KUKA KRL program: MyProgram_311().src

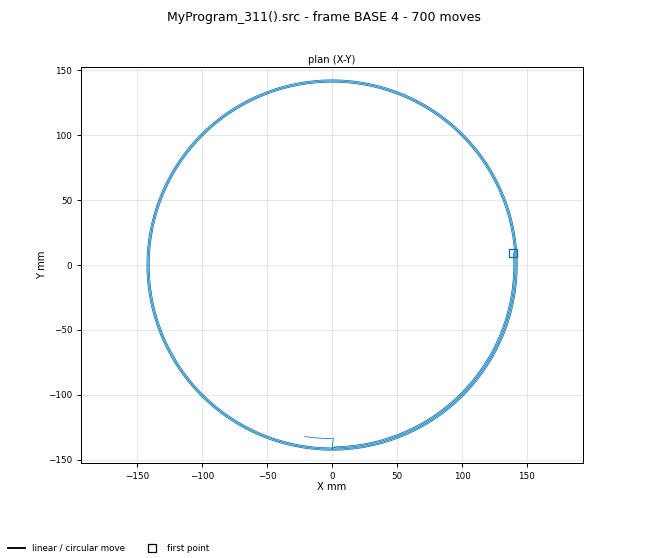
[picture p0: tool path of MyProgram_311().src in frame BASE 4, 700 of 700 moves have a stored position in this frame; points joined in program order, loops and branches not executed]
&ACCESS RVP
&REL 1
&PARAM TEMPLATE = C:\KRC\Roboter\Template\vorgabe
&PARAM EDITMASK = *
DEF MyProgram_311()
; ---- Setting reference (Base) ----
$BASE = BASE_DATA[4]

; --------------------------
; ---- Setting tool (TCP) ----
$TOOL = TOOL_DATA[3]
; --------------------------

$VEL.CP = VEL_APROX_PRINT
Startdeposition()
$VEL.CP = VEL_PRINT
LIN {X 139.5556,Y 9.3465,Z 182,A 6.1945,B 4.3682,C 0.2186,E1 4.5332,E2 446.7738} C_DIS
LIN {X 139.7636,Y 5.3586,Z 182,A 4.7306,B 4.3681,C 0.221,E1 4.5334,E2 448.2166} C_DIS
LIN {X 139.863,Y 1.0803,Z 182,A 3.0816,B 4.3679,C 0.2246,E1 4.5334,E2 449.8533} C_DIS
LIN {X 139.8455,Y -2.4148,Z 182,A 1.6288,B 4.3677,C 0.229,E1 4.5334,E2 451.3099} C_DIS
LIN {X 139.7039,Y -6.743,Z 182,A -0.0934,B 4.3674,C 0.2333,E1 4.5332,E2 453.0267} C_DIS
LIN {X 139.4575,Y -10.6969,Z 182,A -1.7087,B 4.3672,C 0.2378,E1 4.5329,E2 454.6422} C_DIS
LIN {X 139.0946,Y -14.6738,Z 182,A -3.2274,B 4.367,C 0.2409,E1 4.5325,E2 456.1468} C_DIS
LIN {X 138.7184,Y -17.8838,Z 182,A -4.5556,B 4.3668,C 0.2447,E1 4.5321,E2 457.4766} C_DIS
LIN {X 138.1883,Y -21.5997,Z 182,A -5.9216,B 4.3667,C 0.2468,E1 4.5315,E2 458.8215} C_DIS
LIN {X 137.1011,Y -27.6739,Z 182,A -8.4598,B 4.3663,C 0.254,E1 4.5302,E2 461.363} C_DIS
LIN {X 136.3972,Y -30.9569,Z 182,A -9.732,B 4.3661,C 0.2565,E1 4.5295,E2 462.6228} C_DIS
LIN {X 135.1669,Y -35.95,Z 182,A -11.6103,B 4.366,C 0.2593,E1 4.5282,E2 464.4729} C_DIS
LIN {X 133.3888,Y -42.0731,Z 182,A -14.3818,B 4.3654,C 0.2686,E1 4.526,E2 467.2676} C_DIS
LIN {X 132.1888,Y -45.7009,Z 182,A -15.8575,B 4.3652,C 0.2716,E1 4.5247,E2 468.7328} C_DIS
LIN {X 131.0744,Y -48.8061,Z 182,A -17.1041,B 4.3651,C 0.2739,E1 4.5235,E2 469.9668} C_DIS
LIN {X 129.9588,Y -51.7063,Z 182,A -18.4546,B 4.3648,C 0.2783,E1 4.5221,E2 471.3286} C_DIS
LIN {X 128.6386,Y -54.9087,Z 182,A -19.8601,B 4.3646,C 0.2819,E1 4.5206,E2 472.7336} C_DIS
LIN {X 127.1217,Y -58.3322,Z 182,A -21.2882,B 4.3644,C 0.2845,E1 4.519,E2 474.1489} C_DIS
LIN {X 125.7052,Y -61.327,Z 182,A -22.6522,B 4.3642,C 0.2881,E1 4.5173,E2 475.515} C_DIS
LIN {X 123.9954,Y -64.7123,Z 182,A -24.1146,B 4.364,C 0.2909,E1 4.5155,E2 476.9667} C_DIS
LIN {X 121.8931,Y -68.5935,Z 182,A -25.947,B 4.3637,C 0.2958,E1 4.513,E2 478.804} C_DIS
LIN {X 119.5124,Y -72.6628,Z 182,A -28.2329,B 4.363,C 0.3051,E1 4.5096,E2 481.138} C_DIS
LIN {X 117.0621,Y -76.5483,Z 182,A -29.6908,B 4.363,C 0.3043,E1 4.5075,E2 482.5419} C_DIS
LIN {X 114.3471,Y -80.5465,Z 182,A -31.6337,B 4.3628,C 0.3086,E1 4.5044,E2 484.4817} C_DIS
LIN {X 112.2761,Y -83.4091,Z 182,A -33.5934,B 4.3621,C 0.3184,E1 4.5011,E2 486.5099} C_DIS
LIN {X 108.7982,Y -87.8973,Z 182,A -35.2386,B 4.3623,C 0.3151,E1 4.4983,E2 488.0676} C_DIS
LIN {X 105.9724,Y -91.2843,Z 182,A -37.4172,B 4.3617,C 0.3238,E1 4.4943,E2 490.2968} C_DIS
LIN {X 102.9688,Y -94.6595,Z 182,A -38.9115,B 4.3617,C 0.3234,E1 4.4916,E2 491.7457} C_DIS
LIN {X 99.538,Y -98.2618,Z 182,A -40.8482,B 4.3615,C 0.3264,E1 4.4878,E2 493.6707} C_DIS
LIN {X 96.3702,Y -101.3701,Z 182,A -42.5691,B 4.3613,C 0.3289,E1 4.4844,E2 495.3802} C_DIS
LIN {X 93.176,Y -104.3133,Z 182,A -44.299,B 4.3611,C 0.3319,E1 4.4808,E2 497.105} C_DIS
LIN {X 89.7656,Y -107.262,Z 182,A -46.1268,B 4.3608,C 0.3352,E1 4.4769,E2 498.9318} C_DIS
LIN {X 86.198,Y -110.1496,Z 182,A -47.8249,B 4.3608,C 0.3365,E1 4.4733,E2 500.6072} C_DIS
LIN {X 83.8613,Y -111.9394,Z 182,A -49.0987,B 4.3605,C 0.3394,E1 4.4704,E2 501.8911} C_DIS
LIN {X 78.9883,Y -115.4291,Z 182,A -51.5583,B 4.3601,C 0.3437,E1 4.4648,E2 504.3532} C_DIS
LIN {X 76.295,Y -117.2266,Z 182,A -53.2496,B 4.3596,C 0.3503,E1 4.4607,E2 506.094} C_DIS
LIN {X 72.5505,Y -119.5803,Z 182,A -54.3551,B 4.3601,C 0.3448,E1 4.4583,E2 507.1069} C_DIS
LIN {X 67.227,Y -122.6523,Z 182,A -57.1169,B 4.3595,C 0.3515,E1 4.4515,E2 509.9034} C_DIS
LIN {X 63.5857,Y -124.5765,Z 182,A -58.5717,B 4.3595,C 0.3511,E1 4.448,E2 511.3284} C_DIS
LIN {X 60.5652,Y -126.0729,Z 182,A -60.0389,B 4.3593,C 0.354,E1 4.4443,E2 512.8082} C_DIS
LIN {X 57.3664,Y -127.5602,Z 182,A -61.391,B 4.3593,C 0.3548,E1 4.4409,E2 514.1489} C_DIS
LIN {X 54.213,Y -128.9321,Z 182,A -62.8205,B 4.3591,C 0.3568,E1 4.4372,E2 515.5822} C_DIS
LIN {X 50.9804,Y -130.2442,Z 182,A -64.1651,B 4.3591,C 0.3575,E1 4.4337,E2 516.9165} C_DIS
LIN {X 47.7376,Y -131.4674,Z 182,A -65.6245,B 4.3589,C 0.3595,E1 4.4299,E2 518.3822} C_DIS
LIN {X 44.4095,Y -132.6285,Z 182,A -67.1062,B 4.3587,C 0.3615,E1 4.426,E2 519.8699} C_DIS
LIN {X 41.0102,Y -133.7185,Z 182,A -68.4928,B 4.3587,C 0.362,E1 4.4223,E2 521.2473} C_DIS
LIN {X 37.9473,Y -134.6201,Z 182,A -69.7052,B 4.3587,C 0.3622,E1 4.4191,E2 522.4478} C_DIS
LIN {X 34.2391,Y -135.6104,Z 182,A -71.6562,B 4.3582,C 0.3677,E1 4.4136,E2 524.4505} C_DIS
LIN {X 29.2302,Y -136.7778,Z 182,A -73.4098,B 4.3584,C 0.3654,E1 4.409,E2 526.1581} C_DIS
LIN {X 23.4061,Y -137.8942,Z 182,A -75.738,B 4.3584,C 0.3659,E1 4.4027,E2 528.4743} C_DIS
LIN {X 19.0292,Y -138.5677,Z 182,A -77.8353,B 4.358,C 0.3699,E1 4.3967,E2 530.6106} C_DIS
LIN {X 15.027,Y -139.0566,Z 182,A -79.3975,B 4.358,C 0.3697,E1 4.3924,E2 532.1618} C_DIS
LIN {X 10.8973,Y -139.4429,Z 182,A -81.106,B 4.358,C 0.3705,E1 4.3877,E2 533.8725} C_DIS
LIN {X 6.9643,Y -139.6928,Z 182,A -82.6912,B 4.358,C 0.3707,E1 4.3832,E2 535.4545} C_DIS
LIN {X 2.5889,Y -139.8426,Z 182,A -84.4714,B 4.358,C 0.3709,E1 4.3783,E2 537.2339} C_DIS
LIN {X 2.5889,Y -139.8426,Z 182,A -84.4714,B 4.358,C 0.3709,E1 4.3783,E2 537.2339} C_DIS
Enddeposition()
LIN {X 1.0035,Y -140.7616,Z 182,A -84.5459,B 4.3128,C 0.3663,E1 4.3327,E2 537.2758} C_DIS
Startdeposition()
$VEL.CP = VEL_PRINT
LIN {X 4.1947,Y -140.7055,Z 182,A -83.0241,B 4.313,C 0.3637,E1 4.3371,E2 535.7232} C_DIS
LIN {X 8.4297,Y -140.5153,Z 182,A -81.3313,B 4.313,C 0.3635,E1 4.3418,E2 534.0339} C_DIS
LIN {X 12.0807,Y -140.2485,Z 182,A -79.8862,B 4.313,C 0.3635,E1 4.3458,E2 532.5942} C_DIS
LIN {X 15.6538,Y -139.8958,Z 182,A -78.4155,B 4.313,C 0.3627,E1 4.3499,E2 531.1214} C_DIS
LIN {X 21.7686,Y -139.0744,Z 182,A -75.9054,B 4.3132,C 0.3614,E1 4.3569,E2 528.6101} C_DIS
LIN {X 25.7531,Y -138.3934,Z 182,A -74.2127,B 4.3133,C 0.3599,E1 4.3615,E2 526.91} C_DIS
LIN {X 29.5156,Y -137.6385,Z 182,A -72.6715,B 4.3133,C 0.359,E1 4.3657,E2 525.3706} C_DIS
LIN {X 33.4498,Y -136.7363,Z 182,A -71.1692,B 4.3133,C 0.3593,E1 4.3698,E2 523.8865} C_DIS
LIN {X 36.5552,Y -135.9385,Z 182,A -69.7439,B 4.3136,C 0.3568,E1 4.3737,E2 522.4439} C_DIS
LIN {X 41.4818,Y -134.5169,Z 182,A -67.7824,B 4.3136,C 0.3563,E1 4.3789,E2 520.4982} C_DIS
LIN {X 44.766,Y -133.4599,Z 182,A -66.3864,B 4.3137,C 0.3549,E1 4.3826,E2 519.1023} C_DIS
LIN {X 48.3681,Y -132.1983,Z 182,A -64.8799,B 4.3138,C 0.3538,E1 4.3865,E2 517.6013} C_DIS
LIN {X 51.4087,Y -131.0449,Z 182,A -63.5613,B 4.3139,C 0.3524,E1 4.39,E2 516.2824} C_DIS
LIN {X 54.4767,Y -129.7989,Z 182,A -62.2082,B 4.3141,C 0.3507,E1 4.3935,E2 514.9276} C_DIS
LIN {X 57.7378,Y -128.3816,Z 182,A -60.7873,B 4.3141,C 0.3491,E1 4.3971,E2 513.5092} C_DIS
LIN {X 61.0166,Y -126.8563,Z 182,A -59.3503,B 4.3143,C 0.3476,E1 4.4007,E2 512.0759} C_DIS
LIN {X 64.2712,Y -125.239,Z 182,A -57.9029,B 4.3144,C 0.3459,E1 4.4043,E2 510.6317} C_DIS
LIN {X 67.2412,Y -123.6715,Z 182,A -56.2495,B 4.3149,C 0.3405,E1 4.4085,E2 508.9383} C_DIS
LIN {X 70.2583,Y -121.9829,Z 182,A -54.9598,B 4.3149,C 0.3398,E1 4.4116,E2 507.6636} C_DIS
LIN {X 74.8899,Y -119.1955,Z 182,A -53.001,B 4.3149,C 0.3392,E1 4.4161,E2 505.736} C_DIS
LIN {X 78.4114,Y -116.909,Z 182,A -50.8592,B 4.3156,C 0.3311,E1 4.4213,E2 503.5337} C_DIS
LIN {X 82.0265,Y -114.4012,Z 182,A -49.4942,B 4.3154,C 0.3332,E1 4.4243,E2 502.2254} C_DIS
LIN {X 85.449,Y -111.8679,Z 182,A -47.8119,B 4.3156,C 0.3307,E1 4.428,E2 500.5486} C_DIS
LIN {X 88.8686,Y -109.1715,Z 182,A -46.0808,B 4.3159,C 0.3279,E1 4.4318,E2 498.8218} C_DIS
LIN {X 92.2336,Y -106.3443,Z 182,A -44.3097,B 4.3161,C 0.3247,E1 4.4355,E2 497.0515} C_DIS
LIN {X 95.5139,Y -103.4078,Z 182,A -42.5311,B 4.3163,C 0.3213,E1 4.4392,E2 495.2734} C_DIS
LIN {X 98.8564,Y -100.2175,Z 182,A -40.6973,B 4.3166,C 0.318,E1 4.4429,E2 493.4443} C_DIS
LIN {X 102.055,Y -96.9583,Z 182,A -38.5045,B 4.3172,C 0.3099,E1 4.4472,E2 491.2045} C_DIS
LIN {X 105.1058,Y -93.6422,Z 182,A -37.3641,B 4.3168,C 0.3147,E1 4.4492,E2 490.1566} C_DIS
LIN {X 108.3519,Y -89.8657,Z 182,A -35.1583,B 4.3173,C 0.3079,E1 4.4532,E2 487.925} C_DIS
LIN {X 112.1364,Y -85.0962,Z 182,A -32.6312,B 4.3178,C 0.3016,E1 4.4575,E2 485.3891} C_DIS
LIN {X 116.9021,Y -78.4217,Z 182,A -29.6507,B 4.318,C 0.2983,E1 4.4623,E2 482.4542} C_DIS
LIN {X 120.7242,Y -72.4002,Z 182,A -26.7535,B 4.3185,C 0.2912,E1 4.4666,E2 479.5555} C_DIS
LIN {X 122.5931,Y -69.1878,Z 182,A -25.1638,B 4.3188,C 0.2865,E1 4.4688,E2 477.9542} C_DIS
LIN {X 124.7296,Y -65.2531,Z 182,A -23.5005,B 4.319,C 0.2839,E1 4.4709,E2 476.3106} C_DIS
LIN {X 126.4028,Y -61.9505,Z 182,A -22.0299,B 4.3192,C 0.2805,E1 4.4728,E2 474.8437} C_DIS
LIN {X 127.8752,Y -58.8507,Z 182,A -20.675,B 4.3194,C 0.2774,E1 4.4743,E2 473.4931} C_DIS
LIN {X 129.3099,Y -55.6276,Z 182,A -19.2888,B 4.3196,C 0.2743,E1 4.4759,E2 472.1125} C_DIS
LIN {X 130.5822,Y -52.5709,Z 182,A -17.97,B 4.3198,C 0.2711,E1 4.4773,E2 470.7963} C_DIS
LIN {X 131.8258,Y -49.3698,Z 182,A -16.5883,B 4.32,C 0.2675,E1 4.4787,E2 469.4156} C_DIS
LIN {X 133.0706,Y -45.9097,Z 182,A -15.1591,B 4.3202,C 0.2644,E1 4.48,E2 467.9943} C_DIS
LIN {X 134.1721,Y -42.5836,Z 182,A -13.5517,B 4.3206,C 0.2581,E1 4.4814,E2 466.3614} C_DIS
LIN {X 136.0007,Y -36.322,Z 182,A -10.8431,B 4.321,C 0.2501,E1 4.4834,E2 463.6435} C_DIS
LIN {X 136.9727,Y -32.4689,Z 182,A -9.7672,B 4.3209,C 0.2528,E1 4.4841,E2 462.6387} C_DIS
LIN {X 137.5669,Y -29.8472,Z 182,A -7.7789,B 4.3217,C 0.2379,E1 4.4853,E2 460.5298} C_DIS
LIN {X 138.7895,Y -23.5179,Z 182,A -6.228,B 4.3214,C 0.2448,E1 4.486,E2 459.1204} C_DIS
LIN {X 139.3977,Y -19.5929,Z 182,A -4.467,B 4.3217,C 0.2383,E1 4.4867,E2 457.3391} C_DIS
LIN {X 139.9332,Y -15.3061,Z 182,A -2.7578,B 4.322,C 0.234,E1 4.4873,E2 455.6351} C_DIS
LIN {X 140.3029,Y -11.4371,Z 182,A -1.2902,B 4.3221,C 0.231,E1 4.4876,E2 454.1814} C_DIS
LIN {X 140.521,Y -8.3358,Z 182,A -0.0362,B 4.3223,C 0.2276,E1 4.4879,E2 452.9281} C_DIS
LIN {X 140.7039,Y -4.2549,Z 182,A 1.6616,B 4.3226,C 0.2224,E1 4.488,E2 451.2244} C_DIS
LIN {X 140.7701,Y -0.1592,Z 182,A 3.1572,B 4.3226,C 0.2199,E1 4.488,E2 449.7503} C_DIS
LIN {X 140.7346,Y 3.1471,Z 182,A 4.6254,B 4.323,C 0.2145,E1 4.488,E2 448.2651} C_DIS
LIN {X 140.5902,Y 7.0668,Z 182,A 6.0508,B 4.323,C 0.2122,E1 4.4878,E2 446.861} C_DIS
LIN {X 140.3777,Y 10.4737,Z 182,A 7.3856,B 4.3232,C 0.209,E1 4.4876,E2 445.5325} C_DIS
LIN {X 140.018,Y 14.5186,Z 182,A 9.7771,B 4.3239,C 0.1947,E1 4.4869,E2 443.042} C_DIS
LIN {X 139.2272,Y 20.7812,Z 182,A 11.4394,B 4.3237,C 0.1994,E1 4.4863,E2 441.4984} C_DIS
LIN {X 138.7977,Y 23.4691,Z 182,A 12.566,B 4.3238,C 0.196,E1 4.4857,E2 440.3685} C_DIS
LIN {X 138.2105,Y 26.7099,Z 182,A 14.4089,B 4.3243,C 0.1857,E1 4.4847,E2 438.4585} C_DIS
LIN {X 137.1859,Y 31.5521,Z 182,A 15.8637,B 4.3243,C 0.1874,E1 4.4839,E2 437.0765} C_DIS
LIN {X 136.2457,Y 35.4009,Z 182,A 17.3501,B 4.3243,C 0.1847,E1 4.4829,E2 435.6057} C_DIS
LIN {X 135.3426,Y 38.7107,Z 182,A 18.931,B 4.3246,C 0.1785,E1 4.4817,E2 433.9998} C_DIS
LIN {X 134.0511,Y 42.9623,Z 182,A 20.4982,B 4.3246,C 0.1767,E1 4.4804,E2 432.4633} C_DIS
LIN {X 132.8883,Y 46.4356,Z 182,A 21.8914,B 4.3248,C 0.1739,E1 4.4791,E2 431.082} C_DIS
LIN {X 131.8874,Y 49.2054,Z 182,A 23.5596,B 4.3251,C 0.1647,E1 4.4774,E2 429.3517} C_DIS
LIN {X 130.1998,Y 53.5169,Z 182,A 24.8803,B 4.3251,C 0.167,E1 4.4761,E2 428.104} C_DIS
LIN {X 128.92,Y 56.5293,Z 182,A 26.1907,B 4.3251,C 0.1638,E1 4.4747,E2 426.7958} C_DIS
LIN {X 127.624,Y 59.3939,Z 182,A 27.464,B 4.3253,C 0.1606,E1 4.4732,E2 425.5227} C_DIS
LIN {X 126.0079,Y 62.7509,Z 182,A 28.92,B 4.3254,C 0.1575,E1 4.4714,E2 424.0739} C_DIS
LIN {X 124.1359,Y 66.3803,Z 182,A 30.6357,B 4.3256,C 0.1526,E1 4.4692,E2 422.3506} C_DIS
LIN {X 120.9487,Y 72.0235,Z 182,A 32.8923,B 4.3256,C 0.1509,E1 4.4661,E2 420.1425} C_DIS
LIN {X 119.5449,Y 74.3303,Z 182,A 34.2434,B 4.3258,C 0.1451,E1 4.4641,E2 418.7584} C_DIS
LIN {X 117.0756,Y 78.1618,Z 182,A 36.0299,B 4.326,C 0.1415,E1 4.4614,E2 416.9802} C_DIS
LIN {X 114.7222,Y 81.5777,Z 182,A 37.6874,B 4.326,C 0.1379,E1 4.4587,E2 415.3261} C_DIS
LIN {X 112.1161,Y 85.1241,Z 182,A 39.4657,B 4.3262,C 0.134,E1 4.4557,E2 413.549} C_DIS
LIN {X 108.7195,Y 89.4211,Z 182,A 41.7328,B 4.3264,C 0.1286,E1 4.4517,E2 411.2764} C_DIS
LIN {X 105.3023,Y 93.4208,Z 182,A 43.7256,B 4.3264,C 0.1258,E1 4.4481,E2 409.3023} C_DIS
LIN {X 102.4492,Y 96.5408,Z 182,A 45.391,B 4.3265,C 0.1228,E1 4.445,E2 407.6436} C_DIS
LIN {X 99.1559,Y 99.9204,Z 182,A 47.6585,B 4.3268,C 0.1147,E1 4.4404,E2 405.331} C_DIS
LIN {X 95.9178,Y 103.0324,Z 182,A 49.2458,B 4.3268,C 0.114,E1 4.4372,E2 403.7745} C_DIS
LIN {X 93.3927,Y 105.3272,Z 182,A 50.098,B 4.3267,C 0.1177,E1 4.4356,E2 402.9911} C_DIS
LIN {X 91.4403,Y 107.0269,Z 182,A 51.4759,B 4.3268,C 0.1119,E1 4.4326,E2 401.5716} C_DIS
LIN {X 88.5315,Y 109.4449,Z 182,A 52.9487,B 4.3268,C 0.1099,E1 4.4294,E2 400.1071} C_DIS
LIN {X 84.9273,Y 112.2647,Z 182,A 54.7573,B 4.3269,C 0.1072,E1 4.4254,E2 398.3054} C_DIS
LIN {X 80.2164,Y 115.6778,Z 182,A 57.0121,B 4.327,C 0.1045,E1 4.4203,E2 396.0649} C_DIS
LIN {X 77.0128,Y 117.8354,Z 182,A 58.6644,B 4.327,C 0.1011,E1 4.4165,E2 394.4023} C_DIS
LIN {X 73.1718,Y 120.2581,Z 182,A 60.4691,B 4.3271,C 0.0987,E1 4.4122,E2 392.6033} C_DIS
LIN {X 69.2179,Y 122.5762,Z 182,A 62.3151,B 4.3272,C 0.0962,E1 4.4077,E2 390.7598} C_DIS
LIN {X 65.0034,Y 124.8607,Z 182,A 64.133,B 4.3272,C 0.095,E1 4.4033,E2 388.959} C_DIS
LIN {X 60.9382,Y 126.8937,Z 182,A 65.7866,B 4.3272,C 0.0948,E1 4.3992,E2 387.3305} C_DIS
LIN {X 58.695,Y 127.9472,Z 182,A 66.9052,B 4.3272,C 0.0923,E1 4.3963,E2 386.198} C_DIS
LIN {X 55.373,Y 129.42,Z 182,A 68.4385,B 4.3273,C 0.09,E1 4.3924,E2 384.6581} C_DIS
LIN {X 52.2758,Y 130.7012,Z 182,A 69.7157,B 4.3273,C 0.0894,E1 4.3891,E2 383.3921} C_DIS
LIN {X 49.0523,Y 131.9448,Z 182,A 71.1661,B 4.3273,C 0.0874,E1 4.3853,E2 381.9364} C_DIS
LIN {X 43.284,Y 133.9474,Z 182,A 73.9988,B 4.3275,C 0.0813,E1 4.3777,E2 379.0598} C_DIS
LIN {X 39.3705,Y 135.1497,Z 182,A 75.2711,B 4.3275,C 0.084,E1 4.3744,E2 377.8381} C_DIS
LIN {X 35.239,Y 136.2867,Z 182,A 77.0415,B 4.3275,C 0.0824,E1 4.3696,E2 376.0649} C_DIS
LIN {X 32.0185,Y 137.0794,Z 182,A 78.3632,B 4.3275,C 0.0817,E1 4.366,E2 374.7471} C_DIS
LIN {X 28.1546,Y 137.9232,Z 182,A 79.9564,B 4.3275,C 0.0808,E1 4.3617,E2 373.1564} C_DIS
LIN {X 24.58,Y 138.6051,Z 182,A 81.361,B 4.3275,C 0.0808,E1 4.3579,E2 371.762} C_DIS
LIN {X 19.5931,Y 139.3977,Z 182,A 83.3695,B 4.3275,C 0.0802,E1 4.3523,E2 369.7601} C_DIS
LIN {X 16.4005,Y 139.8092,Z 182,A 84.6892,B 4.3275,C 0.0796,E1 4.3487,E2 368.4396} C_DIS
LIN {X 12.902,Y 140.1762,Z 182,A 86.2243,B 4.3275,C 0.078,E1 4.3444,E2 366.892} C_DIS
LIN {X 8.7111,Y 140.4979,Z 182,A 87.865,B 4.3275,C 0.0783,E1 4.3398,E2 365.2608} C_DIS
LIN {X 5.2551,Y 140.6698,Z 182,A 89.2678,B 4.3275,C 0.0781,E1 4.3359,E2 363.8593} C_DIS
LIN {X 1.0534,Y 140.7641,Z 182,A 90.9753,B 4.3275,C 0.0779,E1 4.3311,E2 362.1529} C_DIS
LIN {X -2.6113,Y 140.7438,Z 182,A 92.4194,B 4.3275,C 0.0783,E1 4.3271,E2 360.7155} C_DIS
LIN {X -6.0927,Y 140.6371,Z 182,A 93.9852,B 4.3275,C 0.077,E1 4.3227,E2 359.1317} C_DIS
LIN {X -11.6011,Y 140.289,Z 182,A 96.1482,B 4.3275,C 0.078,E1 4.3167,E2 356.9802} C_DIS
LIN {X -15.7871,Y 139.8815,Z 182,A 97.9546,B 4.3275,C 0.0775,E1 4.3116,E2 355.1628} C_DIS
LIN {X -19.6297,Y 139.3925,Z 182,A 99.8377,B 4.3276,C 0.0752,E1 4.3063,E2 353.2415} C_DIS
LIN {X -23.679,Y 138.7626,Z 182,A 101.262,B 4.3276,C 0.0781,E1 4.3025,E2 351.8491} C_DIS
LIN {X -31.0191,Y 137.3077,Z 182,A 103.9816,B 4.3275,C 0.0826,E1 4.2952,E2 349.1726} C_DIS
LIN {X -34.988,Y 136.3503,Z 182,A 106.2207,B 4.3275,C 0.0785,E1 4.2889,E2 346.8614} C_DIS
LIN {X -38.835,Y 135.3065,Z 182,A 107.424,B 4.3275,C 0.0833,E1 4.2858,E2 345.7123} C_DIS
LIN {X -41.5917,Y 134.4833,Z 182,A 108.6405,B 4.3275,C 0.0838,E1 4.2825,E2 344.4907} C_DIS
LIN {X -44.8359,Y 133.4366,Z 182,A 110.0436,B 4.3275,C 0.0848,E1 4.2788,E2 343.0865} C_DIS
LIN {X -48.4249,Y 132.1778,Z 182,A 112.1415,B 4.3275,C 0.0815,E1 4.2731,E2 340.9198} C_DIS
LIN {X -52.6259,Y 130.5601,Z 182,A 113.1511,B 4.3273,C 0.0903,E1 4.2708,E2 340.0157} C_DIS
LIN {X -56.3123,Y 129.0139,Z 182,A 115.1353,B 4.3273,C 0.089,E1 4.2656,E2 337.9876} C_DIS
LIN {X -60.2781,Y 127.2091,Z 182,A 117.0888,B 4.3273,C 0.0895,E1 4.2606,E2 336.0124} C_DIS
LIN {X -64.3155,Y 125.2165,Z 182,A 118.886,B 4.3273,C 0.0921,E1 4.2561,E2 334.221} C_DIS
LIN {X -68.5617,Y 122.9449,Z 182,A 120.8737,B 4.3273,C 0.0944,E1 4.2512,E2 332.2314} C_DIS
LIN {X -72.1351,Y 120.8822,Z 182,A 122.4835,B 4.3272,C 0.0973,E1 4.2474,E2 330.6316} C_DIS
LIN {X -74.649,Y 119.3466,Z 182,A 123.7999,B 4.3272,C 0.0981,E1 4.2442,E2 329.3012} C_DIS
LIN {X -78.5385,Y 116.8241,Z 182,A 125.6989,B 4.3271,C 0.1009,E1 4.2398,E2 327.402} C_DIS
LIN {X -82.5812,Y 114.0014,Z 182,A 128.0452,B 4.3271,C 0.1014,E1 4.2344,E2 325.014} C_DIS
LIN {X -85.6695,Y 111.6993,Z 182,A 129.7639,B 4.3271,C 0.1029,E1 4.2305,E2 323.2772} C_DIS
LIN {X -89.1843,Y 108.9135,Z 182,A 130.9992,B 4.3269,C 0.1106,E1 4.228,E2 322.1186} C_DIS
LIN {X -92.0514,Y 106.5015,Z 182,A 133.146,B 4.3269,C 0.1086,E1 4.2233,E2 319.8936} C_DIS
LIN {X -95.2287,Y 103.67,Z 182,A 134.2874,B 4.3267,C 0.1164,E1 4.2211,E2 318.8291} C_DIS
LIN {X -99.1991,Y 99.8774,Z 182,A 136.8145,B 4.3267,C 0.1185,E1 4.2159,E2 316.2666} C_DIS
LIN {X -105.2455,Y 93.4851,Z 182,A 141.0681,B 4.3266,C 0.1209,E1 4.2077,E2 311.9298} C_DIS
LIN {X -108.702,Y 89.4429,Z 182,A 142.7173,B 4.3263,C 0.1294,E1 4.2049,E2 310.3487} C_DIS
LIN {X -111.9487,Y 85.3433,Z 182,A 145.061,B 4.3263,C 0.1325,E1 4.2008,E2 307.9792} C_DIS
LIN {X -115.369,Y 80.6602,Z 182,A 147.3588,B 4.3261,C 0.1384,E1 4.1971,E2 305.6915} C_DIS
LIN {X -117.9284,Y 76.8695,Z 182,A 149.2782,B 4.3259,C 0.1423,E1 4.1942,E2 303.7662} C_DIS
LIN {X -120.4175,Y 72.9082,Z 182,A 151.2028,B 4.3258,C 0.1468,E1 4.1913,E2 301.8404} C_DIS
LIN {X -122.6596,Y 69.0695,Z 182,A 153.0643,B 4.3256,C 0.1508,E1 4.1887,E2 299.9738} C_DIS
LIN {X -126.3141,Y 62.1302,Z 182,A 156.0282,B 4.3253,C 0.1604,E1 4.185,E2 297.0419} C_DIS
LIN {X -128.7149,Y 56.9925,Z 182,A 158.6577,B 4.3252,C 0.1642,E1 4.1819,E2 294.3732} C_DIS
LIN {X -131.5073,Y 50.2192,Z 182,A 161.7059,B 4.3249,C 0.1715,E1 4.1786,E2 291.3191} C_DIS
LIN {X -133.1148,Y 45.7821,Z 182,A 163.6801,B 4.3247,C 0.1763,E1 4.1768,E2 289.3396} C_DIS
LIN {X -134.126,Y 42.7279,Z 182,A 165.0836,B 4.3246,C 0.1792,E1 4.1756,E2 287.925} C_DIS
LIN {X -135.1535,Y 39.3576,Z 182,A 166.5277,B 4.3244,C 0.183,E1 4.1744,E2 286.4807} C_DIS
LIN {X -136.071,Y 36.0582,Z 182,A 168.0261,B 4.3243,C 0.1861,E1 4.1733,E2 284.9699} C_DIS
LIN {X -137.0318,Y 32.2237,Z 182,A 169.7755,B 4.3241,C 0.1896,E1 4.1722,E2 283.2036} C_DIS
LIN {X -138.1052,Y 27.2574,Z 182,A 172.2071,B 4.324,C 0.1929,E1 4.1708,E2 280.7263} C_DIS
LIN {X -138.8042,Y 23.4301,Z 182,A 173.788,B 4.3238,C 0.1974,E1 4.17,E2 279.1469} C_DIS
LIN {X -139.3704,Y 19.7842,Z 182,A 174.9794,B 4.3235,C 0.2037,E1 4.1696,E2 277.9972} C_DIS
LIN {X -139.8676,Y 15.8995,Z 182,A 177.1105,B 4.3235,C 0.2045,E1 4.1689,E2 275.797} C_DIS
LIN {X -140.2885,Y 11.6068,Z 182,A 178.4569,B 4.3231,C 0.2123,E1 4.1686,E2 274.5055} C_DIS
LIN {X -140.5305,Y 8.1822,Z 182,A 179.8327,B 4.3229,C 0.2163,E1 4.1683,E2 273.1336} C_DIS
LIN {X -140.6805,Y 4.9818,Z 182,A -178.6444,B 4.3228,C 0.2186,E1 4.1681,E2 271.5831} C_DIS
LIN {X -140.7496,Y -2.2652,Z 182,A -174.8219,B 4.3226,C 0.221,E1 4.1682,E2 267.6476} C_DIS
LIN {X -140.494,Y -8.7754,Z 182,A -172.9378,B 4.322,C 0.2337,E1 4.1685,E2 265.8667} C_DIS
LIN {X -139.938,Y -15.2621,Z 182,A -170.1308,B 4.3216,C 0.2401,E1 4.1692,E2 263.0409} C_DIS
LIN {X -139.1595,Y -21.2188,Z 182,A -167.9046,B 4.3211,C 0.2485,E1 4.1701,E2 260.8451} C_DIS
LIN {X -138.2294,Y -26.6114,Z 182,A -165.4201,B 4.3209,C 0.2529,E1 4.1713,E2 258.3283} C_DIS
LIN {X -137.5648,Y -29.8567,Z 182,A -164.0321,B 4.3207,C 0.2564,E1 4.1721,E2 256.9359} C_DIS
LIN {X -136.8756,Y -32.8719,Z 182,A -162.6476,B 4.3205,C 0.2589,E1 4.173,E2 255.5355} C_DIS
LIN {X -135.9716,Y -36.4308,Z 182,A -161.1579,B 4.3203,C 0.2631,E1 4.174,E2 254.0474} C_DIS
LIN {X -135.0179,Y -39.8207,Z 182,A -159.6706,B 4.3201,C 0.2666,E1 4.1752,E2 252.5538} C_DIS
LIN {X -134.018,Y -43.0658,Z 182,A -158.2589,B 4.3199,C 0.27,E1 4.1764,E2 251.1388} C_DIS
LIN {X -132.9527,Y -46.2498,Z 182,A -155.7202,B 4.3201,C 0.2654,E1 4.1789,E2 248.4443} C_DIS
LIN {X -130.1779,Y -53.5694,Z 182,A -153.5661,B 4.3192,C 0.2811,E1 4.181,E2 246.4302} C_DIS
LIN {X -128.7244,Y -56.9714,Z 182,A -151.8106,B 4.319,C 0.2831,E1 4.183,E2 244.6421} C_DIS
LIN {X -126.8774,Y -60.9723,Z 182,A -150.1387,B 4.3187,C 0.2885,E1 4.1849,E2 242.9873} C_DIS
LIN {X -125.3084,Y -64.135,Z 182,A -148.6642,B 4.3184,C 0.2918,E1 4.1868,E2 241.5083} C_DIS
LIN {X -120.3498,Y -73.0202,Z 182,A -144.4927,B 4.3178,C 0.3017,E1 4.1926,E2 237.3349} C_DIS
LIN {X -117.7957,Y -77.0734,Z 182,A -142.3698,B 4.3175,C 0.305,E1 4.1958,E2 235.1898} C_DIS
LIN {X -115.4224,Y -80.5835,Z 182,A -140.5483,B 4.3173,C 0.3082,E1 4.1987,E2 233.3559} C_DIS
LIN {X -112.5242,Y -84.5834,Z 182,A -138.4695,B 4.317,C 0.3121,E1 4.2021,E2 231.2685} C_DIS
LIN {X -109.7715,Y -88.1265,Z 182,A -136.5849,B 4.3168,C 0.3156,E1 4.2054,E2 229.3766} C_DIS
LIN {X -106.8942,Y -91.5954,Z 182,A -134.6856,B 4.3165,C 0.3189,E1 4.2088,E2 227.4691} C_DIS
LIN {X -103.8445,Y -95.0389,Z 182,A -132.7652,B 4.3163,C 0.3224,E1 4.2124,E2 225.5426} C_DIS
LIN {X -100.6514,Y -98.414,Z 182,A -130.8875,B 4.316,C 0.3262,E1 4.2161,E2 223.6671} C_DIS
LIN {X -97.6591,Y -101.3844,Z 182,A -129.142,B 4.3158,C 0.3292,E1 4.2196,E2 221.9179} C_DIS
LIN {X -94.5514,Y -104.2881,Z 182,A -127.3536,B 4.3155,C 0.3319,E1 4.2233,E2 220.122} C_DIS
LIN {X -91.3093,Y -107.1383,Z 182,A -125.5426,B 4.3153,C 0.3346,E1 4.2271,E2 218.304} C_DIS
LIN {X -87.8447,Y -109.997,Z 182,A -123.7,B 4.3151,C 0.3376,E1 4.2311,E2 216.4597} C_DIS
LIN {X -82.2896,Y -114.2127,Z 182,A -121.069,B 4.3146,C 0.3439,E1 4.2369,E2 213.8569} C_DIS
LIN {X -78.4105,Y -116.9096,Z 182,A -118.8047,B 4.3146,C 0.3439,E1 4.2422,E2 211.5465} C_DIS
LIN {X -74.2689,Y -119.5831,Z 182,A -116.7932,B 4.3144,C 0.3466,E1 4.247,E2 209.5343} C_DIS
LIN {X -70.2353,Y -121.9963,Z 182,A -114.843,B 4.3142,C 0.3489,E1 4.2517,E2 207.579} C_DIS
LIN {X -66.4767,Y -124.0841,Z 182,A -113.2188,B 4.3139,C 0.3521,E1 4.2556,E2 205.9718} C_DIS
LIN {X -63.0467,Y -125.8616,Z 182,A -111.5866,B 4.3139,C 0.3535,E1 4.2597,E2 204.3314} C_DIS
LIN {X -60.3186,Y -127.1897,Z 182,A -110.3032,B 4.3138,C 0.3544,E1 4.263,E2 203.0412} C_DIS
LIN {X -56.7147,Y -128.8392,Z 182,A -108.6877,B 4.3136,C 0.356,E1 4.2671,E2 201.4253} C_DIS
LIN {X -54.0102,Y -129.9937,Z 182,A -107.4542,B 4.3136,C 0.3569,E1 4.2703,E2 200.1865} C_DIS
LIN {X -50.6515,Y -131.3392,Z 182,A -105.9171,B 4.3135,C 0.3576,E1 4.2743,E2 198.6404} C_DIS
LIN {X -45.9387,Y -133.0605,Z 182,A -103.5461,B 4.3136,C 0.3562,E1 4.2807,E2 196.2242} C_DIS
LIN {X -42.2276,Y -134.2858,Z 182,A -102.4566,B 4.3131,C 0.3621,E1 4.2834,E2 195.2026} C_DIS
LIN {X -37.1862,Y -135.769,Z 182,A -100.1698,B 4.3131,C 0.3621,E1 4.2896,E2 192.8953} C_DIS
LIN {X -34.3211,Y -136.5197,Z 182,A -98.9829,B 4.3131,C 0.363,E1 4.2928,E2 191.7105} C_DIS
LIN {X -31.1721,Y -137.2728,Z 182,A -97.5933,B 4.3131,C 0.363,E1 4.2966,E2 190.3108} C_DIS
LIN {X -27.6185,Y -138.0323,Z 182,A -96.1507,B 4.313,C 0.364,E1 4.3005,E2 188.8727} C_DIS
LIN {X -23.5776,Y -138.7796,Z 182,A -94.4135,B 4.313,C 0.364,E1 4.3053,E2 187.1262} C_DIS
LIN {X -19.9733,Y -139.3434,Z 182,A -92.9444,B 4.313,C 0.3645,E1 4.3094,E2 185.6586} C_DIS
LIN {X -16.3072,Y -139.8204,Z 182,A -91.3948,B 4.313,C 0.3644,E1 4.3137,E2 184.1024} C_DIS
LIN {X -12.0315,Y -140.2527,Z 182,A -89.6971,B 4.3129,C 0.3651,E1 4.3184,E2 182.411} C_DIS
LIN {X -7.9746,Y -140.5433,Z 182,A -87.9153,B 4.3129,C 0.3639,E1 4.3234,E2 180.6114} C_DIS
LIN {X -3.8519,Y -140.7151,Z 182,A -86.3459,B 4.3129,C 0.365,E1 4.3278,E2 179.0562} C_DIS
LIN {X 0.4359,Y -140.7675,Z 182,A -84.5705,B 4.3129,C 0.3644,E1 4.3327,E2 177.2759} C_DIS
LIN {X 0.4359,Y -140.7675,Z 182,A -84.5705,B 4.3129,C 0.3644,E1 4.3327,E2 177.2759} C_DIS
Enddeposition()
LIN {X 1.012,Y -141.6629,Z 182,A -84.5652,B 4.3123,C 0.3691,E1 4.3324,E2 177.3331} C_DIS
Startdeposition()
$VEL.CP = VEL_PRINT
LIN {X -1.7962,Y -141.659,Z 182,A -86.2004,B 4.3119,C 0.3745,E1 4.3276,E2 179.0371} C_DIS
LIN {X -5.8291,Y -141.5496,Z 182,A -87.7532,B 4.3119,C 0.3737,E1 4.3233,E2 180.5799} C_DIS
LIN {X -9.9926,Y -141.3167,Z 182,A -89.4602,B 4.3119,C 0.3739,E1 4.3185,E2 182.2904} C_DIS
LIN {X -13.7811,Y -140.9974,Z 182,A -90.9429,B 4.3119,C 0.3731,E1 4.3144,E2 183.7662} C_DIS
LIN {X -17.2558,Y -140.6151,Z 182,A -92.5209,B 4.3119,C 0.3745,E1 4.31,E2 185.3671} C_DIS
LIN {X -21.6784,Y -140.0006,Z 182,A -94.2326,B 4.3119,C 0.3731,E1 4.3053,E2 187.0666} C_DIS
LIN {X -25.2898,Y -139.3938,Z 182,A -95.6994,B 4.312,C 0.3724,E1 4.3012,E2 188.532} C_DIS
LIN {X -28.8866,Y -138.6942,Z 182,A -97.1586,B 4.3121,C 0.3716,E1 4.2973,E2 189.9886} C_DIS
LIN {X -32.4597,Y -137.9022,Z 182,A -98.6333,B 4.3121,C 0.3708,E1 4.2932,E2 191.4631} C_DIS
LIN {X -35.3227,Y -137.1955,Z 182,A -99.9996,B 4.3121,C 0.3718,E1 4.2895,E2 192.8532} C_DIS
LIN {X -40.6214,Y -135.7228,Z 182,A -102.9587,B 4.3116,C 0.3771,E1 4.2813,E2 195.9118} C_DIS
LIN {X -46.6366,Y -133.7727,Z 182,A -105.1118,B 4.3121,C 0.3714,E1 4.2757,E2 198.0111} C_DIS
LIN {X -50.5739,Y -132.3366,Z 182,A -106.3862,B 4.3126,C 0.3661,E1 4.2726,E2 199.2291} C_DIS
LIN {X -53.2463,Y -131.2819,Z 182,A -107.6055,B 4.3126,C 0.3655,E1 4.2694,E2 200.4564} C_DIS
LIN {X -56.4002,Y -129.958,Z 182,A -109.0139,B 4.3127,C 0.3644,E1 4.2657,E2 201.8684} C_DIS
LIN {X -59.8237,Y -128.4185,Z 182,A -110.5464,B 4.3128,C 0.3629,E1 4.2618,E2 203.403} C_DIS
LIN {X -63.242,Y -126.7709,Z 182,A -112.0884,B 4.313,C 0.3612,E1 4.258,E2 204.9462} C_DIS
LIN {X -66.9091,Y -124.8751,Z 182,A -114.1075,B 4.3129,C 0.3623,E1 4.2529,E2 207.0125} C_DIS
LIN {X -70.0722,Y -123.128,Z 182,A -115.2894,B 4.3133,C 0.358,E1 4.2501,E2 208.1569} C_DIS
LIN {X -73.7479,Y -120.9628,Z 182,A -117.0886,B 4.3133,C 0.3563,E1 4.2457,E2 209.9661} C_DIS
LIN {X -77.2036,Y -118.7863,Z 182,A -118.7908,B 4.3136,C 0.3544,E1 4.2417,E2 211.6751} C_DIS
LIN {X -81.1298,Y -116.1404,Z 182,A -120.7191,B 4.3138,C 0.3516,E1 4.2373,E2 213.6052} C_DIS
LIN {X -84.5752,Y -113.6557,Z 182,A -122.559,B 4.3139,C 0.3499,E1 4.2331,E2 215.4613} C_DIS
LIN {X -88.1217,Y -110.9287,Z 182,A -124.2896,B 4.3142,C 0.3463,E1 4.2293,E2 217.1812} C_DIS
LIN {X -91.4662,Y -108.1881,Z 182,A -126.1449,B 4.3144,C 0.3441,E1 4.2253,E2 219.0507} C_DIS
LIN {X -94.869,Y -105.2171,Z 182,A -127.9916,B 4.3146,C 0.341,E1 4.2214,E2 220.8998} C_DIS
LIN {X -98.2606,Y -102.0568,Z 182,A -129.9921,B 4.3148,C 0.3385,E1 4.2173,E2 222.9167} C_DIS
LIN {X -102.1511,Y -98.1625,Z 182,A -132.1886,B 4.3152,C 0.334,E1 4.2131,E2 225.1089} C_DIS
LIN {X -105.2705,Y -94.8096,Z 182,A -134.1005,B 4.3154,C 0.3307,E1 4.2094,E2 227.0283} C_DIS
LIN {X -108.3145,Y -91.3162,Z 182,A -136.0176,B 4.3157,C 0.3271,E1 4.2059,E2 228.9507} C_DIS
LIN {X -111.2986,Y -87.654,Z 182,A -137.9184,B 4.316,C 0.323,E1 4.2026,E2 230.8497} C_DIS
LIN {X -113.9757,Y -84.144,Z 182,A -139.8115,B 4.3162,C 0.3198,E1 4.1994,E2 232.7566} C_DIS
LIN {X -116.6929,Y -80.3329,Z 182,A -141.7381,B 4.3165,C 0.3158,E1 4.1963,E2 234.6871} C_DIS
LIN {X -119.3084,Y -76.3943,Z 182,A -143.4793,B 4.317,C 0.3101,E1 4.1937,E2 236.4048} C_DIS
LIN {X -121.0463,Y -73.6104,Z 182,A -145.023,B 4.317,C 0.3086,E1 4.1914,E2 237.9769} C_DIS
LIN {X -123.1808,Y -69.9796,Z 182,A -147.1782,B 4.3171,C 0.3077,E1 4.1883,E2 240.1912} C_DIS
LIN {X -125.184,Y -66.3268,Z 182,A -148.3217,B 4.3177,C 0.2997,E1 4.1869,E2 241.2623} C_DIS
LIN {X -127.2305,Y -62.3103,Z 182,A -150.3949,B 4.3179,C 0.2969,E1 4.1843,E2 243.3679} C_DIS
LIN {X -129.4853,Y -57.478,Z 182,A -152.5763,B 4.3182,C 0.2916,E1 4.1817,E2 245.5516} C_DIS
LIN {X -130.9084,Y -54.1595,Z 182,A -154.1723,B 4.3184,C 0.2888,E1 4.18,E2 247.1649} C_DIS
LIN {X -133.6956,Y -46.859,Z 182,A -157.1737,B 4.319,C 0.2794,E1 4.1771,E2 250.1437} C_DIS
LIN {X -135.0002,Y -42.9537,Z 182,A -159.0424,B 4.3192,C 0.2764,E1 4.1754,E2 252.0384} C_DIS
LIN {X -136.0163,Y -39.6189,Z 182,A -160.501,B 4.3195,C 0.2729,E1 4.1742,E2 253.5026} C_DIS
LIN {X -136.9535,Y -36.2475,Z 182,A -161.9351,B 4.3197,C 0.2692,E1 4.1732,E2 254.9384} C_DIS
LIN {X -137.7439,Y -33.1163,Z 182,A -163.2608,B 4.3199,C 0.2658,E1 4.1723,E2 256.2659} C_DIS
LIN {X -138.4596,Y -29.9839,Z 182,A -164.6267,B 4.3201,C 0.2627,E1 4.1714,E2 257.6397} C_DIS
LIN {X -139.4924,Y -24.739,Z 182,A -166.8953,B 4.3204,C 0.2574,E1 4.1703,E2 259.921} C_DIS
LIN {X -140.4839,Y -18.2872,Z 182,A -169.7652,B 4.3208,C 0.2516,E1 4.1691,E2 262.8194} C_DIS
LIN {X -141.1421,Y -12.2123,Z 182,A -171.9536,B 4.3213,C 0.2427,E1 4.1685,E2 264.9691} C_DIS
LIN {X -141.4151,Y -8.4846,Z 182,A -173.7623,B 4.3213,C 0.2405,E1 4.1681,E2 266.8157} C_DIS
LIN {X -141.5959,Y -4.6083,Z 182,A -175.6892,B 4.3215,C 0.2384,E1 4.1679,E2 268.788} C_DIS
LIN {X -141.6657,Y -1.1317,Z 182,A -176.9137,B 4.3218,C 0.2332,E1 4.1679,E2 269.9879} C_DIS
LIN {X -141.6493,Y 2.3773,Z 182,A -178.3618,B 4.322,C 0.2294,E1 4.1679,E2 271.4387} C_DIS
LIN {X -141.4858,Y 7.2076,Z 182,A 179.6624,B 4.3223,C 0.224,E1 4.1681,E2 273.4159} C_DIS
LIN {X -141.2409,Y 11.0303,Z 182,A 178.0046,B 4.3225,C 0.2203,E1 4.1685,E2 275.0866} C_DIS
LIN {X -140.7426,Y 16.1866,Z 182,A 176.0293,B 4.3228,C 0.2136,E1 4.169,E2 277.0448} C_DIS
LIN {X -140.2446,Y 20.0394,Z 182,A 174.2473,B 4.3229,C 0.2106,E1 4.1697,E2 278.8529} C_DIS
LIN {X -139.6246,Y 23.9905,Z 182,A 171.8481,B 4.3229,C 0.2113,E1 4.1709,E2 281.3514} C_DIS
LIN {X -138.5093,Y 29.7538,Z 182,A 170.4449,B 4.3235,C 0.1982,E1 4.1716,E2 282.6279} C_DIS
LIN {X -137.6814,Y 33.3759,Z 182,A 168.626,B 4.3236,C 0.1962,E1 4.1728,E2 284.4866} C_DIS
LIN {X -136.8496,Y 36.6371,Z 182,A 167.1982,B 4.3238,C 0.1929,E1 4.1738,E2 285.9219} C_DIS
LIN {X -135.9429,Y 39.8695,Z 182,A 165.8716,B 4.3239,C 0.189,E1 4.1748,E2 287.2433} C_DIS
LIN {X -134.9068,Y 43.2462,Z 182,A 164.3153,B 4.3241,C 0.186,E1 4.1761,E2 288.8149} C_DIS
LIN {X -133.7174,Y 46.7959,Z 182,A 162.7224,B 4.3242,C 0.1825,E1 4.1776,E2 290.4167} C_DIS
LIN {X -132.3225,Y 50.6102,Z 182,A 160.7501,B 4.3243,C 0.1804,E1 4.1795,E2 292.43} C_DIS
LIN {X -131.0273,Y 53.8746,Z 182,A 159.6456,B 4.3245,C 0.1745,E1 4.1807,E2 293.4929} C_DIS
LIN {X -129.8523,Y 56.6447,Z 182,A 158.3605,B 4.3247,C 0.1718,E1 4.1821,E2 294.7858} C_DIS
LIN {X -128.3978,Y 59.8684,Z 182,A 156.8575,B 4.3247,C 0.1686,E1 4.1838,E2 296.2969} C_DIS
LIN {X -125.9511,Y 64.8596,Z 182,A 154.4159,B 4.3249,C 0.1643,E1 4.1869,E2 298.7614} C_DIS
LIN {X -123.7349,Y 68.9959,Z 182,A 152.4995,B 4.3251,C 0.1597,E1 4.1895,E2 300.6786} C_DIS
LIN {X -121.4692,Y 72.9109,Z 182,A 150.6129,B 4.3253,C 0.1556,E1 4.1922,E2 302.5711} C_DIS
LIN {X -119.035,Y 76.8206,Z 182,A 148.6992,B 4.3254,C 0.1516,E1 4.195,E2 304.4897} C_DIS
LIN {X -116.4935,Y 80.6223,Z 182,A 146.7816,B 4.3255,C 0.1477,E1 4.1981,E2 306.4144} C_DIS
LIN {X -111.8417,Y 86.9601,Z 182,A 143.8368,B 4.3258,C 0.1389,E1 4.2029,E2 309.3267} C_DIS
LIN {X -108.5113,Y 91.0818,Z 182,A 141.2173,B 4.3258,C 0.1377,E1 4.2076,E2 312.005} C_DIS
LIN {X -104.3446,Y 95.8269,Z 182,A 138.5391,B 4.326,C 0.1332,E1 4.2127,E2 314.6968} C_DIS
LIN {X -102.0664,Y 98.2506,Z 182,A 137.475,B 4.3262,C 0.1285,E1 4.2147,E2 315.7243} C_DIS
LIN {X -99.4844,Y 100.8642,Z 182,A 135.8031,B 4.3262,C 0.1269,E1 4.218,E2 317.4186} C_DIS
LIN {X -96.2113,Y 103.9912,Z 182,A 133.8251,B 4.3262,C 0.1245,E1 4.2221,E2 319.4138} C_DIS
LIN {X -91.6464,Y 108.0349,Z 182,A 131.6225,B 4.3265,C 0.118,E1 4.2266,E2 321.581} C_DIS
LIN {X -88.7972,Y 110.3887,Z 182,A 129.9049,B 4.3265,C 0.1171,E1 4.2304,E2 323.3257} C_DIS
LIN {X -85.3273,Y 113.0921,Z 182,A 127.486,B 4.3265,C 0.119,E1 4.236,E2 325.8235} C_DIS
LIN {X -80.8167,Y 116.3583,Z 182,A 126.2537,B 4.3267,C 0.1075,E1 4.2385,E2 326.9258} C_DIS
LIN {X -76.8206,Y 119.035,Z 182,A 123.609,B 4.3267,C 0.1101,E1 4.2448,E2 329.6574} C_DIS
LIN {X -73.9805,Y 120.82,Z 182,A 122.5293,B 4.3267,C 0.1059,E1 4.2473,E2 330.7014} C_DIS
LIN {X -69.9784,Y 123.1815,Z 182,A 120.8164,B 4.3269,C 0.102,E1 4.2514,E2 332.3918} C_DIS
LIN {X -65.4446,Y 125.6472,Z 182,A 118.5289,B 4.3269,C 0.1009,E1 4.2571,E2 334.7031} C_DIS
LIN {X -62.3937,Y 127.1893,Z 182,A 117.0962,B 4.3269,C 0.0996,E1 4.2607,E2 336.1411} C_DIS
LIN {X -58.864,Y 128.8622,Z 182,A 115.435,B 4.3269,C 0.0985,E1 4.2649,E2 337.8115} C_DIS
LIN {X -55.7117,Y 130.2556,Z 182,A 114.0816,B 4.3269,C 0.0967,E1 4.2684,E2 339.1589} C_DIS
LIN {X -52.4744,Y 131.5931,Z 182,A 112.5465,B 4.3269,C 0.0963,E1 4.2724,E2 340.7079} C_DIS
LIN {X -48.0657,Y 133.2656,Z 182,A 110.6681,B 4.327,C 0.0943,E1 4.2773,E2 342.5815} C_DIS
LIN {X -44.4509,Y 134.5149,Z 182,A 109.1917,B 4.327,C 0.0923,E1 4.2812,E2 344.0481} C_DIS
LIN {X -41.1694,Y 135.5553,Z 182,A 107.7427,B 4.327,C 0.0918,E1 4.285,E2 345.5034} C_DIS
LIN {X -35.3841,Y 137.18,Z 182,A 105.422,B 4.3271,C 0.0891,E1 4.2913,E2 347.8089} C_DIS
LIN {X -30.6942,Y 138.3063,Z 182,A 103.2134,B 4.3271,C 0.0903,E1 4.2973,E2 350.0489} C_DIS
LIN {X -26.6822,Y 139.1336,Z 182,A 101.2012,B 4.3271,C 0.0927,E1 4.303,E2 352.1046} C_DIS
LIN {X -22.2932,Y 139.9054,Z 182,A 99.8202,B 4.3271,C 0.0882,E1 4.3067,E2 353.4319} C_DIS
LIN {X -18.6138,Y 140.4411,Z 182,A 98.3372,B 4.3271,C 0.0875,E1 4.3107,E2 354.9115} C_DIS
LIN {X -14.4799,Y 140.9288,Z 182,A 96.5277,B 4.3271,C 0.0883,E1 4.3158,E2 356.736} C_DIS
LIN {X -9.9836,Y 141.3173,Z 182,A 94.7766,B 4.3271,C 0.0873,E1 4.3207,E2 358.4769} C_DIS
LIN {X -5.1768,Y 141.575,Z 182,A 92.7657,B 4.3271,C 0.0878,E1 4.3263,E2 360.4949} C_DIS
LIN {X -0.754,Y 141.6673,Z 182,A 91.074,B 4.3271,C 0.0869,E1 4.331,E2 362.1736} C_DIS
LIN {X 3.2224,Y 141.6344,Z 182,A 89.3848,B 4.3271,C 0.0879,E1 4.3357,E2 363.8724} C_DIS
LIN {X 7.1399,Y 141.4892,Z 182,A 87.9091,B 4.3271,C 0.0871,E1 4.3398,E2 365.3335} C_DIS
LIN {X 11.2989,Y 141.2192,Z 182,A 86.1713,B 4.3271,C 0.0881,E1 4.3447,E2 367.0773} C_DIS
LIN {X 15.4116,Y 140.8286,Z 182,A 84.5376,B 4.3271,C 0.0883,E1 4.3492,E2 368.7057} C_DIS
LIN {X 19.759,Y 140.2846,Z 182,A 82.7085,B 4.3271,C 0.0897,E1 4.3543,E2 370.5413} C_DIS
LIN {X 24.1923,Y 139.5903,Z 182,A 80.9586,B 4.3271,C 0.09,E1 4.3591,E2 372.2826} C_DIS
LIN {X 28.0823,Y 138.8579,Z 182,A 79.3316,B 4.3271,C 0.0912,E1 4.3635,E2 373.9123} C_DIS
LIN {X 32.0952,Y 137.9866,Z 182,A 77.6991,B 4.3271,C 0.0921,E1 4.368,E2 375.5409} C_DIS
LIN {X 37.0994,Y 136.7263,Z 182,A 75.7455,B 4.3271,C 0.0923,E1 4.3732,E2 377.4771} C_DIS
LIN {X 42.9614,Y 134.9978,Z 182,A 72.7446,B 4.3269,C 0.1,E1 4.3814,E2 380.5441} C_DIS
LIN {X 47.401,Y 133.5053,Z 182,A 71.4414,B 4.327,C 0.0957,E1 4.3847,E2 381.7725} C_DIS
LIN {X 51.1816,Y 132.1003,Z 182,A 69.7584,B 4.327,C 0.0979,E1 4.3891,E2 383.4618} C_DIS
LIN {X 54.8134,Y 130.6353,Z 182,A 68.1893,B 4.327,C 0.0996,E1 4.3931,E2 385.0288} C_DIS
LIN {X 58.5782,Y 128.9932,Z 182,A 66.4315,B 4.3268,C 0.1026,E1 4.3976,E2 386.7987} C_DIS
LIN {X 63.0113,Y 126.8847,Z 182,A 64.1104,B 4.3267,C 0.1089,E1 4.4036,E2 389.1619} C_DIS
LIN {X 67.1548,Y 124.7431,Z 182,A 62.7148,B 4.3267,C 0.1061,E1 4.4069,E2 390.4956} C_DIS
LIN {X 70.886,Y 122.6612,Z 182,A 60.9634,B 4.3267,C 0.1088,E1 4.4111,E2 392.2498} C_DIS
LIN {X 74.6308,Y 120.4196,Z 182,A 59.2564,B 4.3267,C 0.1109,E1 4.4152,E2 393.9495} C_DIS
LIN {X 78.1103,Y 118.1923,Z 182,A 57.5728,B 4.3266,C 0.1137,E1 4.4191,E2 395.6347} C_DIS
LIN {X 81.9696,Y 115.5496,Z 182,A 55.7554,B 4.3266,C 0.1159,E1 4.4233,E2 397.4427} C_DIS
LIN {X 84.6715,Y 113.584,Z 182,A 54.4113,B 4.3264,C 0.1182,E1 4.4263,E2 398.786} C_DIS
LIN {X 88.284,Y 110.7995,Z 182,A 52.6347,B 4.3264,C 0.1207,E1 4.4302,E2 400.5541} C_DIS
LIN {X 92.2457,Y 107.5239,Z 182,A 50.8653,B 4.3264,C 0.1209,E1 4.4339,E2 402.2842} C_DIS
LIN {X 99.5904,Y 100.7594,Z 182,A 46.8838,B 4.3262,C 0.1282,E1 4.4421,E2 406.2592} C_DIS
LIN {X 103.2886,Y 96.9648,Z 182,A 44.5682,B 4.326,C 0.1347,E1 4.4466,E2 408.5974} C_DIS
LIN {X 106.5588,Y 93.3588,Z 182,A 42.8651,B 4.326,C 0.1356,E1 4.4497,E2 410.2668} C_DIS
LIN {X 111.4666,Y 87.4402,Z 182,A 39.6166,B 4.3257,C 0.1442,E1 4.4555,E2 413.5341} C_DIS
LIN {X 114.0867,Y 83.993,Z 182,A 37.8619,B 4.3255,C 0.1483,E1 4.4584,E2 415.2899} C_DIS
LIN {X 116.8032,Y 80.1723,Z 182,A 36.0627,B 4.3255,C 0.1515,E1 4.4613,E2 417.0773} C_DIS
LIN {X 119.0728,Y 76.7623,Z 182,A 34.4366,B 4.3253,C 0.1551,E1 4.4638,E2 418.6999} C_DIS
LIN {X 121.3622,Y 73.0881,Z 182,A 32.7438,B 4.3252,C 0.1586,E1 4.4662,E2 420.386} C_DIS
LIN {X 123.5814,Y 69.2694,Z 182,A 30.9978,B 4.325,C 0.1625,E1 4.4687,E2 422.1275} C_DIS
LIN {X 125.5921,Y 65.5495,Z 182,A 29.3686,B 4.3249,C 0.1658,E1 4.4708,E2 423.7469} C_DIS
LIN {X 127.3445,Y 62.0791,Z 182,A 27.8916,B 4.3248,C 0.1686,E1 4.4726,E2 425.2122} C_DIS
LIN {X 128.6049,Y 59.4204,Z 182,A 26.6785,B 4.3246,C 0.1719,E1 4.474,E2 426.4288} C_DIS
LIN {X 130.3028,Y 55.6027,Z 182,A 25.065,B 4.3246,C 0.1754,E1 4.4758,E2 428.0333} C_DIS
LIN {X 131.7346,Y 52.1222,Z 182,A 23.4949,B 4.3243,C 0.18,E1 4.4775,E2 429.6103} C_DIS
LIN {X 132.817,Y 49.2937,Z 182,A 22.4112,B 4.3243,C 0.1814,E1 4.4785,E2 430.6762} C_DIS
LIN {X 133.9653,Y 46.0809,Z 182,A 21.0749,B 4.3241,C 0.1846,E1 4.4798,E2 432.0076} C_DIS
LIN {X 135.2613,Y 42.1299,Z 182,A 19.2197,B 4.3238,C 0.1914,E1 4.4814,E2 433.8863} C_DIS
LIN {X 136.6014,Y 37.5566,Z 182,A 16.5196,B 4.3231,C 0.2065,E1 4.4835,E2 436.6871} C_DIS
LIN {X 138.4643,Y 29.9623,Z 182,A 14.4291,B 4.3234,C 0.2015,E1 4.4846,E2 438.641} C_DIS
LIN {X 139.285,Y 25.8901,Z 182,A 12.9108,B 4.3233,C 0.2041,E1 4.4854,E2 440.1392} C_DIS
LIN {X 139.8754,Y 22.4861,Z 182,A 11.4059,B 4.323,C 0.2094,E1 4.4861,E2 441.6591} C_DIS
LIN {X 140.4552,Y 18.5062,Z 182,A 9.7124,B 4.3227,C 0.2148,E1 4.4868,E2 443.3624} C_DIS
LIN {X 141.0667,Y 13.0598,Z 182,A 7.6963,B 4.3226,C 0.2185,E1 4.4873,E2 445.3538} C_DIS
LIN {X 141.3982,Y 8.7579,Z 182,A 6.1009,B 4.3224,C 0.2214,E1 4.4876,E2 446.9306} C_DIS
LIN {X 141.5862,Y 4.8913,Z 182,A 4.6432,B 4.3222,C 0.2245,E1 4.4878,E2 448.3753} C_DIS
LIN {X 141.6659,Y 1.0932,Z 182,A 2.9343,B 4.3219,C 0.2311,E1 4.4878,E2 450.1079} C_DIS
LIN {X 141.6035,Y -4.3334,Z 182,A 1.0558,B 4.3218,C 0.2332,E1 4.4878,E2 451.9463} C_DIS
LIN {X 141.4795,Y -7.332,Z 182,A -0.1408,B 4.3216,C 0.2364,E1 4.4876,E2 453.1415} C_DIS
LIN {X 141.282,Y -10.4674,Z 182,A -1.4102,B 4.3214,C 0.24,E1 4.4874,E2 454.4117} C_DIS
LIN {X 140.9794,Y -13.9692,Z 182,A -2.784,B 4.3212,C 0.2433,E1 4.487,E2 455.7803} C_DIS
LIN {X 140.6149,Y -17.2575,Z 182,A -4.1308,B 4.321,C 0.2472,E1 4.4866,E2 457.1292} C_DIS
LIN {X 140.033,Y -21.4689,Z 182,A -5.8409,B 4.3207,C 0.252,E1 4.4859,E2 458.8395} C_DIS
LIN {X 139.3976,Y -25.2689,Z 182,A -7.531,B 4.3204,C 0.258,E1 4.4851,E2 460.5482} C_DIS
LIN {X 138.7614,Y -28.5562,Z 182,A -8.5893,B 4.3204,C 0.258,E1 4.4845,E2 461.5685} C_DIS
LIN {X 137.8414,Y -32.712,Z 182,A -10.321,B 4.3201,C 0.2629,E1 4.4834,E2 463.3029} C_DIS
LIN {X 136.812,Y -36.7781,Z 182,A -11.8539,B 4.3199,C 0.2654,E1 4.4824,E2 464.8154} C_DIS
LIN {X 135.0855,Y -42.6867,Z 182,A -14.1412,B 4.3197,C 0.2696,E1 4.4806,E2 467.0778} C_DIS
LIN {X 134.3367,Y -44.9861,Z 182,A -15.2482,B 4.3194,C 0.2739,E1 4.4796,E2 468.2028} C_DIS
LIN {X 133.0181,Y -48.7523,Z 182,A -16.8331,B 4.3191,C 0.2779,E1 4.4781,E2 469.7853} C_DIS
LIN {X 131.5358,Y -52.6166,Z 182,A -18.5027,B 4.3189,C 0.2823,E1 4.4764,E2 471.4556} C_DIS
LIN {X 129.9854,Y -56.3367,Z 182,A -20.0279,B 4.3187,C 0.2852,E1 4.4747,E2 472.9682} C_DIS
LIN {X 128.4331,Y -59.7921,Z 182,A -21.4892,B 4.3185,C 0.2883,E1 4.4731,E2 474.4214} C_DIS
LIN {X 126.975,Y -62.8282,Z 182,A -22.8306,B 4.3182,C 0.2916,E1 4.4714,E2 475.7611} C_DIS
LIN {X 125.3274,Y -66.0536,Z 182,A -24.2167,B 4.3181,C 0.2943,E1 4.4696,E2 477.138} C_DIS
LIN {X 123.2941,Y -69.7805,Z 182,A -26.0202,B 4.3177,C 0.2997,E1 4.4672,E2 478.9546} C_DIS
LIN {X 120.4733,Y -74.5446,Z 182,A -28.192,B 4.3174,C 0.3044,E1 4.4641,E2 481.1192} C_DIS
LIN {X 118.0447,Y -78.3338,Z 182,A -29.9115,B 4.3171,C 0.3075,E1 4.4615,E2 482.8268} C_DIS
LIN {X 115.6624,Y -81.8097,Z 182,A -31.5988,B 4.3169,C 0.3114,E1 4.4588,E2 484.5132} C_DIS
LIN {X 111.9989,Y -86.7573,Z 182,A -34.0598,B 4.3165,C 0.3168,E1 4.4546,E2 486.9725} C_DIS
LIN {X 109.0116,Y -90.4824,Z 182,A -35.9033,B 4.3162,C 0.32,E1 4.4514,E2 488.8059} C_DIS
LIN {X 106.019,Y -93.9712,Z 182,A -37.6825,B 4.316,C 0.3231,E1 4.4482,E2 490.5759} C_DIS
LIN {X 102.7945,Y -97.4885,Z 182,A -39.4539,B 4.3158,C 0.3253,E1 4.4448,E2 492.3276} C_DIS
LIN {X 100.3787,Y -99.9736,Z 182,A -40.9356,B 4.3155,C 0.3292,E1 4.4419,E2 493.8213} C_DIS
LIN {X 97.1236,Y -103.1387,Z 182,A -42.7338,B 4.3153,C 0.3325,E1 4.4383,E2 495.6159} C_DIS
LIN {X 93.8967,Y -106.0848,Z 182,A -44.491,B 4.315,C 0.3359,E1 4.4346,E2 497.3732} C_DIS
LIN {X 90.5708,Y -108.9385,Z 182,A -46.1981,B 4.3148,C 0.3385,E1 4.431,E2 499.073} C_DIS
LIN {X 87.1467,Y -111.697,Z 182,A -47.951,B 4.3146,C 0.3414,E1 4.4272,E2 500.8238} C_DIS
LIN {X 83.5609,Y -114.4042,Z 182,A -49.7602,B 4.3143,C 0.3446,E1 4.4231,E2 502.6335} C_DIS
LIN {X 79.9853,Y -116.9315,Z 182,A -51.4595,B 4.3142,C 0.3467,E1 4.4192,E2 504.3245} C_DIS
LIN {X 76.511,Y -119.2337,Z 182,A -53.1051,B 4.314,C 0.349,E1 4.4154,E2 505.966} C_DIS
LIN {X 72.8545,Y -121.5028,Z 182,A -54.7966,B 4.3138,C 0.3512,E1 4.4114,E2 507.6523} C_DIS
LIN {X 67.4394,Y -124.5902,Z 182,A -57.3462,B 4.3135,C 0.3553,E1 4.4052,E2 510.2077} C_DIS
LIN {X 63.9236,Y -126.4275,Z 182,A -58.8344,B 4.3135,C 0.3562,E1 4.4015,E2 511.6813} C_DIS
LIN {X 60.8052,Y -127.9563,Z 182,A -60.1909,B 4.3133,C 0.3575,E1 4.3981,E2 513.0322} C_DIS
LIN {X 57.7773,Y -129.3515,Z 182,A -61.5132,B 4.3132,C 0.359,E1 4.3947,E2 514.3521} C_DIS
LIN {X 54.0787,Y -130.9421,Z 182,A -63.1387,B 4.313,C 0.3609,E1 4.3905,E2 515.9783} C_DIS
LIN {X 50.4278,Y -132.3922,Z 182,A -64.6633,B 4.313,C 0.362,E1 4.3866,E2 517.4954} C_DIS
LIN {X 47.6321,Y -133.4219,Z 182,A -65.8625,B 4.3128,C 0.3633,E1 4.3834,E2 518.6946} C_DIS
LIN {X 44.3039,Y -134.5639,Z 182,A -67.4211,B 4.3126,C 0.3662,E1 4.3793,E2 520.2725} C_DIS
LIN {X 39.5716,Y -136.0302,Z 182,A -69.2934,B 4.3126,C 0.3667,E1 4.3743,E2 522.1283} C_DIS
LIN {X 36.0747,Y -136.9996,Z 182,A -70.9094,B 4.3123,C 0.3696,E1 4.3699,E2 523.7655} C_DIS
LIN {X 30.7289,Y -138.2986,Z 182,A -72.9141,B 4.3123,C 0.3689,E1 4.3645,E2 525.7416} C_DIS
LIN {X 25.8482,Y -139.2926,Z 182,A -74.89,B 4.3123,C 0.3698,E1 4.3591,E2 527.7135} C_DIS
LIN {X 22.4028,Y -139.8884,Z 182,A -76.4634,B 4.312,C 0.3724,E1 4.3547,E2 529.3094} C_DIS
LIN {X 18.2139,Y -140.4935,Z 182,A -78.0685,B 4.312,C 0.3722,E1 4.3503,E2 530.9009} C_DIS
LIN {X 13.7493,Y -141.0005,Z 182,A -79.8463,B 4.312,C 0.3725,E1 4.3454,E2 532.6743} C_DIS
LIN {X 10.1988,Y -141.3016,Z 182,A -81.3133,B 4.312,C 0.3733,E1 4.3413,E2 534.1456} C_DIS
LIN {X 5.7802,Y -141.5515,Z 182,A -83.0814,B 4.312,C 0.3736,E1 4.3363,E2 535.9116} C_DIS
LIN {X 2.2725,Y -141.651,Z 182,A -84.5019,B 4.312,C 0.3739,E1 4.3324,E2 537.3331} C_DIS
LIN {X 2.2725,Y -141.651,Z 182,A -84.5019,B 4.312,C 0.3739,E1 4.3324,E2 537.3331} C_DIS
Enddeposition()
LIN {X 1.0202,Y -142.5636,Z 182,A -84.547,B 4.3123,C 0.3715,E1 4.3324,E2 537.3468} C_DIS
Startdeposition()
$VEL.CP = VEL_PRINT
LIN {X 4.6622,Y -142.4962,Z 182,A -82.7363,B 4.3126,C 0.3676,E1 4.3377,E2 535.4877} C_DIS
LIN {X 8.7545,Y -142.3016,Z 182,A -81.2385,B 4.3125,C 0.3687,E1 4.3418,E2 534.0096} C_DIS
LIN {X 12.2387,Y -142.0445,Z 182,A -79.7657,B 4.3126,C 0.3674,E1 4.3459,E2 532.5264} C_DIS
LIN {X 16.3065,Y -141.6362,Z 182,A -78.2455,B 4.3126,C 0.368,E1 4.3501,E2 531.0224} C_DIS
LIN {X 19.7974,Y -141.1898,Z 182,A -76.7926,B 4.3126,C 0.3669,E1 4.3541,E2 529.5634} C_DIS
LIN {X 23.2514,Y -140.6619,Z 182,A -75.5834,B 4.3126,C 0.3682,E1 4.3574,E2 528.3803} C_DIS
LIN {X 26.1067,Y -140.1614,Z 182,A -74.1096,B 4.3129,C 0.3641,E1 4.3616,E2 526.8631} C_DIS
LIN {X 30.1106,Y -139.3545,Z 182,A -72.6409,B 4.3129,C 0.3648,E1 4.3655,E2 525.4173} C_DIS
LIN {X 34.772,Y -138.2654,Z 182,A -70.6907,B 4.3129,C 0.363,E1 4.3708,E2 523.4623} C_DIS
LIN {X 37.8484,Y -137.4559,Z 182,A -69.2947,B 4.3132,C 0.3606,E1 4.3747,E2 522.0491} C_DIS
LIN {X 41.9348,Y -136.2638,Z 182,A -67.6745,B 4.3132,C 0.36,E1 4.379,E2 520.4404} C_DIS
LIN {X 46.3958,Y -134.8103,Z 182,A -65.8925,B 4.3132,C 0.3592,E1 4.3836,E2 518.6714} C_DIS
LIN {X 49.6854,Y -133.6329,Z 182,A -64.5064,B 4.3134,C 0.3579,E1 4.3873,E2 517.2869} C_DIS
LIN {X 52.945,Y -132.3754,Z 182,A -63.1222,B 4.3135,C 0.3565,E1 4.3909,E2 515.9044} C_DIS
LIN {X 56.7185,Y -130.8025,Z 182,A -61.4341,B 4.3137,C 0.354,E1 4.3952,E2 514.2089} C_DIS
LIN {X 60.9506,Y -128.8859,Z 182,A -59.5909,B 4.3139,C 0.3518,E1 4.3999,E2 512.3676} C_DIS
LIN {X 64.6038,Y -127.0929,Z 182,A -58.0487,B 4.3139,C 0.3507,E1 4.4037,E2 510.8371} C_DIS
LIN {X 68.0075,Y -125.3072,Z 182,A -56.4738,B 4.3142,C 0.3481,E1 4.4076,E2 509.257} C_DIS
LIN {X 71.8111,Y -123.1673,Z 182,A -54.6951,B 4.3144,C 0.3451,E1 4.4119,E2 507.4734} C_DIS
LIN {X 75.7972,Y -120.7549,Z 182,A -52.8632,B 4.3146,C 0.3427,E1 4.4163,E2 505.6456} C_DIS
LIN {X 79.4553,Y -118.3799,Z 182,A -51.1379,B 4.3148,C 0.3401,E1 4.4203,E2 503.9228} C_DIS
LIN {X 83.2875,Y -115.716,Z 182,A -49.2947,B 4.3151,C 0.3372,E1 4.4245,E2 502.0826} C_DIS
LIN {X 87.0295,Y -112.9285,Z 182,A -47.4651,B 4.3153,C 0.3344,E1 4.4286,E2 500.2578} C_DIS
LIN {X 90.4468,Y -110.2101,Z 182,A -45.8533,B 4.3153,C 0.3329,E1 4.432,E2 498.6643} C_DIS
LIN {X 93.5707,Y -107.5704,Z 182,A -44.1496,B 4.3157,C 0.329,E1 4.4357,E2 496.9509} C_DIS
LIN {X 97.041,Y -104.4504,Z 182,A -42.3234,B 4.3159,C 0.3259,E1 4.4394,E2 495.13} C_DIS
LIN {X 100.1948,Y -101.4297,Z 182,A -40.5918,B 4.3162,C 0.3226,E1 4.4429,E2 493.4001} C_DIS
LIN {X 103.4628,Y -98.0937,Z 182,A -38.7616,B 4.3164,C 0.3192,E1 4.4464,E2 491.5747} C_DIS
LIN {X 106.6153,Y -94.6577,Z 182,A -36.9375,B 4.3167,C 0.3157,E1 4.4498,E2 489.7559} C_DIS
LIN {X 109.6546,Y -91.1194,Z 182,A -35.1173,B 4.3169,C 0.3123,E1 4.4531,E2 487.9415} C_DIS
LIN {X 112.418,Y -87.6881,Z 182,A -33.3789,B 4.3172,C 0.3086,E1 4.4561,E2 486.2061} C_DIS
LIN {X 115.2228,Y -83.9682,Z 182,A -31.5612,B 4.3175,C 0.305,E1 4.4591,E2 484.3942} C_DIS
LIN {X 117.8929,Y -80.176,Z 182,A -29.7455,B 4.3177,C 0.3012,E1 4.462,E2 482.5835} C_DIS
LIN {X 120.2886,Y -76.5352,Z 182,A -28.0962,B 4.3179,C 0.2982,E1 4.4645,E2 480.9467} C_DIS
LIN {X 122.429,Y -73.0613,Z 182,A -26.4684,B 4.3182,C 0.2943,E1 4.4668,E2 479.3191} C_DIS
LIN {X 124.7589,Y -69.0075,Z 182,A -24.686,B 4.3184,C 0.2909,E1 4.4692,E2 477.5484} C_DIS
LIN {X 126.8233,Y -65.1332,Z 182,A -22.9518,B 4.3187,C 0.2868,E1 4.4715,E2 475.8167} C_DIS
LIN {X 128.6384,Y -61.4686,Z 182,A -21.489,B 4.3188,C 0.2849,E1 4.4732,E2 474.3772} C_DIS
LIN {X 129.9842,Y -58.5705,Z 182,A -20.1185,B 4.3191,C 0.2804,E1 4.4748,E2 472.9938} C_DIS
LIN {X 131.7166,Y -54.5633,Z 182,A -18.4729,B 4.3193,C 0.2772,E1 4.4766,E2 471.3616} C_DIS
LIN {X 133.23,Y -50.7609,Z 182,A -16.8818,B 4.3196,C 0.2735,E1 4.4782,E2 469.7764} C_DIS
LIN {X 134.4348,Y -47.4789,Z 182,A -15.5148,B 4.3198,C 0.2703,E1 4.4795,E2 468.4134} C_DIS
LIN {X 135.6232,Y -43.966,Z 182,A -13.9791,B 4.3201,C 0.2656,E1 4.4809,E2 466.8703} C_DIS
LIN {X 136.9394,Y -39.6743,Z 182,A -12.2521,B 4.3203,C 0.2617,E1 4.4822,E2 465.1523} C_DIS
LIN {X 138.0179,Y -35.7471,Z 182,A -10.7343,B 4.3205,C 0.2588,E1 4.4833,E2 463.6493} C_DIS
LIN {X 138.8514,Y -32.3574,Z 182,A -9.4642,B 4.3205,C 0.2566,E1 4.4841,E2 462.396} C_DIS
LIN {X 139.4794,Y -29.5323,Z 182,A -8.1397,B 4.3209,C 0.2513,E1 4.4849,E2 461.0488} C_DIS
LIN {X 140.2722,Y -25.499,Z 182,A -6.8183,B 4.3209,C 0.251,E1 4.4856,E2 459.7707} C_DIS
LIN {X 140.7637,Y -22.6406,Z 182,A -5.514,B 4.3212,C 0.2459,E1 4.4862,E2 458.4469} C_DIS
LIN {X 141.3528,Y -18.5944,Z 182,A -4.0825,B 4.3213,C 0.2441,E1 4.4868,E2 457.0426} C_DIS
LIN {X 141.7024,Y -15.7169,Z 182,A -2.797,B 4.3216,C 0.2392,E1 4.4872,E2 455.7399} C_DIS
LIN {X 142.1251,Y -11.2855,Z 182,A -1.1,B 4.3218,C 0.2354,E1 4.4876,E2 454.054} C_DIS
LIN {X 142.3393,Y -8.1431,Z 182,A 0.2697,B 4.3221,C 0.2304,E1 4.4878,E2 452.6694} C_DIS
LIN {X 142.5052,Y -4.3391,Z 182,A 1.5234,B 4.3221,C 0.2298,E1 4.488,E2 451.4517} C_DIS
LIN {X 142.5695,Y -0.7791,Z 182,A 3.0604,B 4.3224,C 0.2243,E1 4.488,E2 449.8995} C_DIS
LIN {X 142.5281,Y 3.5124,Z 182,A 4.6996,B 4.3226,C 0.2205,E1 4.488,E2 448.2705} C_DIS
LIN {X 142.3986,Y 7.0045,Z 182,A 6.0505,B 4.3228,C 0.2173,E1 4.4878,E2 446.9259} C_DIS
LIN {X 142.1842,Y 10.4909,Z 182,A 7.4032,B 4.3229,C 0.214,E1 4.4875,E2 445.5791} C_DIS
LIN {X 141.8264,Y 14.5646,Z 182,A 9.0167,B 4.3231,C 0.2097,E1 4.4871,E2 443.9684} C_DIS
LIN {X 141.4972,Y 17.4711,Z 182,A 10.2523,B 4.3233,C 0.2056,E1 4.4867,E2 442.724} C_DIS
LIN {X 140.9378,Y 21.5171,Z 182,A 11.7298,B 4.3234,C 0.2032,E1 4.4861,E2 441.2674} C_DIS
LIN {X 140.4728,Y 24.3778,Z 182,A 12.8627,B 4.3236,C 0.2004,E1 4.4856,E2 440.1381} C_DIS
LIN {X 139.7107,Y 28.4121,Z 182,A 14.4632,B 4.3237,C 0.1964,E1 4.4847,E2 438.5431} C_DIS
LIN {X 138.8374,Y 32.4188,Z 182,A 16.1783,B 4.324,C 0.191,E1 4.4836,E2 436.8182} C_DIS
LIN {X 137.8499,Y 36.3845,Z 182,A 17.6356,B 4.324,C 0.1889,E1 4.4826,E2 435.3845} C_DIS
LIN {X 136.932,Y 39.6997,Z 182,A 18.985,B 4.3242,C 0.1856,E1 4.4816,E2 434.0387} C_DIS
LIN {X 135.9124,Y 43.0605,Z 182,A 20.3486,B 4.3244,C 0.1824,E1 4.4805,E2 432.6807} C_DIS
LIN {X 134.8159,Y 46.3796,Z 182,A 21.71,B 4.3244,C 0.1792,E1 4.4793,E2 431.3244} C_DIS
LIN {X 133.6383,Y 49.6709,Z 182,A 23.0775,B 4.3246,C 0.1759,E1 4.478,E2 429.9611} C_DIS
LIN {X 132.3726,Y 52.9519,Z 182,A 24.4414,B 4.3248,C 0.1728,E1 4.4766,E2 428.603} C_DIS
LIN {X 130.801,Y 56.722,Z 182,A 26.1015,B 4.3249,C 0.1683,E1 4.4748,E2 426.9396} C_DIS
LIN {X 128.8854,Y 60.9518,Z 182,A 27.9173,B 4.3251,C 0.1641,E1 4.4726,E2 425.1297} C_DIS
LIN {X 127.0936,Y 64.6024,Z 182,A 29.4377,B 4.3251,C 0.1614,E1 4.4708,E2 423.6236} C_DIS
LIN {X 125.3238,Y 67.977,Z 182,A 30.9863,B 4.3253,C 0.1574,E1 4.4687,E2 422.0721} C_DIS
LIN {X 123.1736,Y 71.8003,Z 182,A 32.749,B 4.3255,C 0.153,E1 4.4663,E2 420.3087} C_DIS
LIN {X 120.7592,Y 75.7903,Z 182,A 34.5666,B 4.3256,C 0.1492,E1 4.4636,E2 418.4979} C_DIS
LIN {X 118.3815,Y 79.4528,Z 182,A 36.2744,B 4.3258,C 0.1456,E1 4.461,E2 416.7958} C_DIS
LIN {X 115.7226,Y 83.2784,Z 182,A 38.1058,B 4.3258,C 0.1417,E1 4.458,E2 414.9691} C_DIS
LIN {X 112.9304,Y 87.027,Z 182,A 39.9357,B 4.326,C 0.1381,E1 4.455,E2 413.145} C_DIS
LIN {X 110.1899,Y 90.4716,Z 182,A 41.647,B 4.326,C 0.1349,E1 4.452,E2 411.4409} C_DIS
LIN {X 107.1887,Y 94.0081,Z 182,A 43.3684,B 4.3262,C 0.1326,E1 4.4489,E2 409.7377} C_DIS
LIN {X 104.4517,Y 97.0396,Z 182,A 45.0573,B 4.3262,C 0.1285,E1 4.4457,E2 408.0421} C_DIS
LIN {X 101.4298,Y 100.1947,Z 182,A 46.7972,B 4.3264,C 0.1251,E1 4.4423,E2 406.3041} C_DIS
LIN {X 98.2783,Y 103.2874,Z 182,A 48.454,B 4.3264,C 0.123,E1 4.439,E2 404.6624} C_DIS
LIN {X 95.0815,Y 106.2371,Z 182,A 50.0148,B 4.3264,C 0.1218,E1 4.4358,E2 403.1257} C_DIS
LIN {X 92.4652,Y 108.522,Z 182,A 51.5822,B 4.3266,C 0.1172,E1 4.4324,E2 401.5357} C_DIS
LIN {X 89.0875,Y 111.3121,Z 182,A 53.2717,B 4.3266,C 0.1148,E1 4.4288,E2 399.8553} C_DIS
LIN {X 85.6306,Y 113.9926,Z 182,A 54.9834,B 4.3267,C 0.1122,E1 4.425,E2 398.1495} C_DIS
LIN {X 82.0464,Y 116.5986,Z 182,A 56.7656,B 4.3268,C 0.1092,E1 4.421,E2 396.3671} C_DIS
LIN {X 78.228,Y 119.1941,Z 182,A 58.5379,B 4.3268,C 0.1072,E1 4.4169,E2 394.6055} C_DIS
LIN {X 74.7947,Y 121.3781,Z 182,A 60.1645,B 4.3269,C 0.1047,E1 4.413,E2 392.9801} C_DIS
LIN {X 71.0307,Y 123.619,Z 182,A 61.9519,B 4.327,C 0.1018,E1 4.4087,E2 391.1892} C_DIS
LIN {X 67.1758,Y 125.7551,Z 182,A 63.7116,B 4.327,C 0.0995,E1 4.4044,E2 389.431} C_DIS
LIN {X 63.2873,Y 127.7537,Z 182,A 65.3618,B 4.327,C 0.0984,E1 4.4003,E2 387.7947} C_DIS
LIN {X 60.1587,Y 129.2567,Z 182,A 66.6799,B 4.3271,C 0.0975,E1 4.397,E2 386.4867} C_DIS
LIN {X 56.7198,Y 130.8019,Z 182,A 68.2705,B 4.3271,C 0.0948,E1 4.3929,E2 384.8865} C_DIS
LIN {X 52.931,Y 132.381,Z 182,A 69.8742,B 4.3271,C 0.0934,E1 4.3888,E2 383.289} C_DIS
LIN {X 48.8908,Y 133.9264,Z 182,A 71.4601,B 4.3271,C 0.0933,E1 4.3847,E2 381.7232} C_DIS
LIN {X 45.7749,Y 135.0242,Z 182,A 72.8342,B 4.3272,C 0.0915,E1 4.381,E2 380.3433} C_DIS
LIN {X 41.9202,Y 136.2682,Z 182,A 74.5403,B 4.3272,C 0.0891,E1 4.3765,E2 378.6274} C_DIS
LIN {X 37.2535,Y 137.6182,Z 182,A 76.3245,B 4.3272,C 0.0893,E1 4.3717,E2 376.8654} C_DIS
LIN {X 34.0499,Y 138.4462,Z 182,A 77.7027,B 4.3273,C 0.0878,E1 4.368,E2 375.4813} C_DIS
LIN {X 31.222,Y 139.1107,Z 182,A 78.85,B 4.3273,C 0.0872,E1 4.3648,E2 374.3369} C_DIS
LIN {X 27.2245,Y 139.9477,Z 182,A 80.4902,B 4.3273,C 0.0862,E1 4.3604,E2 372.6973} C_DIS
LIN {X 24.3742,Y 140.4735,Z 182,A 81.7744,B 4.3273,C 0.0843,E1 4.3568,E2 371.3981} C_DIS
LIN {X 20.9051,Y 141.0315,Z 182,A 83.1925,B 4.3273,C 0.0835,E1 4.3529,E2 369.9797} C_DIS
LIN {X 17.4408,Y 141.5009,Z 182,A 84.4543,B 4.3273,C 0.0844,E1 4.3494,E2 368.7369} C_DIS
LIN {X 13.9677,Y 141.8851,Z 182,A 85.946,B 4.3274,C 0.083,E1 4.3452,E2 367.2343} C_DIS
LIN {X 9.8942,Y 142.2277,Z 182,A 87.5976,B 4.3274,C 0.0824,E1 4.3406,E2 365.5822} C_DIS
LIN {X 5.2328,Y 142.475,Z 182,A 89.3387,B 4.3274,C 0.0834,E1 4.3358,E2 363.8593} C_DIS
LIN {X 1.0886,Y 142.5669,Z 182,A 91.0104,B 4.3274,C 0.0832,E1 4.3312,E2 362.1875} C_DIS
LIN {X -2.3484,Y 142.5514,Z 182,A 92.4583,B 4.3274,C 0.0825,E1 4.3271,E2 360.7317} C_DIS
LIN {X -7.0191,Y 142.3978,Z 182,A 94.2773,B 4.3274,C 0.0831,E1 4.322,E2 358.9211} C_DIS
LIN {X -10.506,Y 142.1831,Z 182,A 95.6766,B 4.3274,C 0.0833,E1 4.3181,E2 357.5231} C_DIS
LIN {X -14.5731,Y 141.8255,Z 182,A 97.3392,B 4.3274,C 0.0834,E1 4.3135,E2 355.8585} C_DIS
LIN {X -17.4558,Y 141.4991,Z 182,A 98.6149,B 4.3274,C 0.0827,E1 4.3099,E2 354.5693} C_DIS
LIN {X -21.5503,Y 140.9326,Z 182,A 100.1667,B 4.3274,C 0.0843,E1 4.3057,E2 353.0324} C_DIS
LIN {X -24.4137,Y 140.4664,Z 182,A 101.3429,B 4.3274,C 0.0847,E1 4.3024,E2 351.8555} C_DIS
LIN {X -28.4196,Y 139.7092,Z 182,A 103.0423,B 4.3274,C 0.0849,E1 4.2978,E2 350.1492} C_DIS
LIN {X -32.9416,Y 138.7134,Z 182,A 104.8565,B 4.3274,C 0.0864,E1 4.2928,E2 348.342} C_DIS
LIN {X -36.3152,Y 137.8684,Z 182,A 106.264,B 4.3274,C 0.0872,E1 4.289,E2 346.9342} C_DIS
LIN {X -39.7145,Y 136.9277,Z 182,A 107.8054,B 4.3274,C 0.0871,E1 4.2848,E2 345.3777} C_DIS
LIN {X -44.157,Y 135.5622,Z 182,A 109.6599,B 4.3273,C 0.0887,E1 4.2799,E2 343.526} C_DIS
LIN {X -48.0568,Y 134.2271,Z 182,A 111.2509,B 4.3273,C 0.0907,E1 4.2757,E2 341.9445} C_DIS
LIN {X -51.3297,Y 133.0099,Z 182,A 112.669,B 4.3273,C 0.0919,E1 4.272,E2 340.5254} C_DIS
LIN {X -54.5707,Y 131.7135,Z 182,A 114.2082,B 4.3273,C 0.0922,E1 4.268,E2 338.9696} C_DIS
LIN {X -58.8461,Y 129.8609,Z 182,A 116.1046,B 4.3272,C 0.094,E1 4.2632,E2 337.0714} C_DIS
LIN {X -62.7914,Y 127.9984,Z 182,A 117.8285,B 4.3272,C 0.0963,E1 4.2588,E2 335.3525} C_DIS
LIN {X -66.1769,Y 126.2809,Z 182,A 119.3068,B 4.3271,C 0.0986,E1 4.2552,E2 333.8814} C_DIS
LIN {X -69.8941,Y 124.2644,Z 182,A 121.1031,B 4.3271,C 0.1,E1 4.2508,E2 332.0739} C_DIS
LIN {X -73.8178,Y 121.9744,Z 182,A 122.9827,B 4.327,C 0.1022,E1 4.2462,E2 330.1887} C_DIS
LIN {X -77.7993,Y 119.4744,Z 182,A 124.8534,B 4.327,C 0.1051,E1 4.2418,E2 328.3218} C_DIS
LIN {X -81.4151,Y 117.0401,Z 182,A 126.6909,B 4.3269,C 0.1071,E1 4.2376,E2 326.4746} C_DIS
LIN {X -85.1949,Y 114.3182,Z 182,A 128.6052,B 4.3269,C 0.1099,E1 4.2333,E2 324.5562} C_DIS
LIN {X -88.867,Y 111.4876,Z 182,A 130.4593,B 4.3267,C 0.1131,E1 4.2292,E2 322.7048} C_DIS
LIN {X -92.2307,Y 108.7214,Z 182,A 132.3059,B 4.3267,C 0.1155,E1 4.2252,E2 320.847} C_DIS
LIN {X -95.7673,Y 105.6193,Z 182,A 134.2236,B 4.3266,C 0.1188,E1 4.2212,E2 318.9274} C_DIS
LIN {X -99.1651,Y 102.4358,Z 182,A 136.1362,B 4.3265,C 0.1221,E1 4.2173,E2 317.0108} C_DIS
LIN {X -102.4438,Y 99.1569,Z 182,A 138.0148,B 4.3264,C 0.1256,E1 4.2136,E2 315.1318} C_DIS
LIN {X -105.0844,Y 96.3541,Z 182,A 139.6421,B 4.3264,C 0.1282,E1 4.2105,E2 313.4954} C_DIS
LIN {X -108.1701,Y 92.8767,Z 182,A 141.5612,B 4.3262,C 0.1318,E1 4.207,E2 311.5713} C_DIS
LIN {X -111.1262,Y 89.3187,Z 182,A 143.4063,B 4.3261,C 0.1359,E1 4.2037,E2 309.7296} C_DIS
LIN {X -113.7974,Y 85.8892,Z 182,A 145.2533,B 4.326,C 0.1391,E1 4.2006,E2 307.8709} C_DIS
LIN {X -116.5652,Y 82.0937,Z 182,A 147.1982,B 4.3258,C 0.143,E1 4.1974,E2 305.9202} C_DIS
LIN {X -119.2566,Y 78.1331,Z 182,A 149.17,B 4.3257,C 0.1472,E1 4.1943,E2 303.9438} C_DIS
LIN {X -121.6848,Y 74.2948,Z 182,A 151.0066,B 4.3256,C 0.1514,E1 4.1916,E2 302.1072} C_DIS
LIN {X -123.766,Y 70.7729,Z 182,A 152.7465,B 4.3254,C 0.1548,E1 4.1892,E2 300.3562} C_DIS
LIN {X -125.8968,Y 66.9084,Z 182,A 154.5521,B 4.3253,C 0.1589,E1 4.1868,E2 298.5478} C_DIS
LIN {X -127.7558,Y 63.283,Z 182,A 156.2215,B 4.3251,C 0.1629,E1 4.1847,E2 296.8755} C_DIS
LIN {X -129.2635,Y 60.144,Z 182,A 157.6013,B 4.325,C 0.1666,E1 4.183,E2 295.4995} C_DIS
LIN {X -130.8032,Y 56.7169,Z 182,A 159.26,B 4.3249,C 0.1694,E1 4.1812,E2 293.8225} C_DIS
LIN {X -132.4937,Y 52.6515,Z 182,A 161.0296,B 4.3247,C 0.1741,E1 4.1793,E2 292.0545} C_DIS
LIN {X -133.845,Y 49.1167,Z 182,A 162.5579,B 4.3245,C 0.1781,E1 4.1778,E2 290.5264} C_DIS
LIN {X -135.0112,Y 45.8139,Z 182,A 164.013,B 4.3244,C 0.1815,E1 4.1765,E2 289.0663} C_DIS
LIN {X -136.2571,Y 41.9564,Z 182,A 165.7989,B 4.3243,C 0.1848,E1 4.175,E2 287.261} C_DIS
LIN {X -137.5642,Y 37.4558,Z 182,A 167.6456,B 4.324,C 0.1902,E1 4.1736,E2 285.4207} C_DIS
LIN {X -138.441,Y 34.0716,Z 182,A 169.1023,B 4.3239,C 0.1937,E1 4.1726,E2 283.9583} C_DIS
LIN {X -139.2267,Y 30.7024,Z 182,A 170.4405,B 4.3237,C 0.1979,E1 4.1717,E2 282.6281} C_DIS
LIN {X -139.953,Y 27.197,Z 182,A 172.0224,B 4.3235,C 0.2009,E1 4.1709,E2 281.0284} C_DIS
LIN {X -140.4786,Y 24.3459,Z 182,A 173.2145,B 4.3234,C 0.204,E1 4.1703,E2 279.8337} C_DIS
LIN {X -141.0316,Y 20.9044,Z 182,A 174.8218,B 4.3233,C 0.2065,E1 4.1696,E2 278.2001} C_DIS
LIN {X -141.4994,Y 17.4533,Z 182,A 176.146,B 4.3231,C 0.211,E1 4.1691,E2 276.887} C_DIS
LIN {X -141.8872,Y 13.9463,Z 182,A 177.6895,B 4.3229,C 0.2141,E1 4.1687,E2 275.3279} C_DIS
LIN {X -142.2286,Y 9.8817,Z 182,A 179.2647,B 4.3227,C 0.2192,E1 4.1683,E2 273.7624} C_DIS
LIN {X -142.4514,Y 5.8383,Z 182,A -179.2011,B 4.3224,C 0.2244,E1 4.1681,E2 272.2418} C_DIS
LIN {X -142.5514,Y 2.3488,Z 182,A -177.5367,B 4.3223,C 0.2266,E1 4.1681,E2 270.5437} C_DIS
LIN {X -142.551,Y -2.3695,Z 182,A -175.5612,B 4.322,C 0.2314,E1 4.1681,E2 268.559} C_DIS
LIN {X -142.3982,Y -7.0114,Z 182,A -173.6901,B 4.3217,C 0.2367,E1 4.1683,E2 266.6887} C_DIS
LIN {X -142.1843,Y -10.4893,Z 182,A -172.2099,B 4.3215,C 0.2401,E1 4.1685,E2 265.1987} C_DIS
LIN {X -141.8202,Y -14.6223,Z 182,A -170.5056,B 4.3213,C 0.2445,E1 4.169,E2 263.4907} C_DIS
LIN {X -141.4916,Y -17.5182,Z 182,A -169.1796,B 4.3212,C 0.2467,E1 4.1695,E2 262.1447} C_DIS
LIN {X -140.9347,Y -21.5367,Z 182,A -167.6209,B 4.3209,C 0.2518,E1 4.1701,E2 260.5967} C_DIS
LIN {X -140.3809,Y -24.8914,Z 182,A -166.3766,B 4.3206,C 0.2564,E1 4.1707,E2 259.3696} C_DIS
LIN {X -139.7133,Y -28.3995,Z 182,A -164.7254,B 4.3205,C 0.2589,E1 4.1716,E2 257.6903} C_DIS
LIN {X -138.8506,Y -32.3609,Z 182,A -162.9169,B 4.3203,C 0.2621,E1 4.1727,E2 255.8589} C_DIS
LIN {X -137.8184,Y -36.5028,Z 182,A -161.3087,B 4.3199,C 0.2676,E1 4.1738,E2 254.266} C_DIS
LIN {X -136.9274,Y -39.7155,Z 182,A -159.7713,B 4.3198,C 0.2698,E1 4.175,E2 252.7028} C_DIS
LIN {X -135.5624,Y -44.1564,Z 182,A -157.9579,B 4.3195,C 0.2752,E1 4.1765,E2 250.8977} C_DIS
LIN {X -134.4295,Y -47.4942,Z 182,A -156.4945,B 4.3192,C 0.2786,E1 4.1778,E2 249.4287} C_DIS
LIN {X -133.2257,Y -50.7726,Z 182,A -154.8956,B 4.3191,C 0.2809,E1 4.1794,E2 247.8043} C_DIS
LIN {X -131.7133,Y -54.5713,Z 182,A -153.2346,B 4.3188,C 0.285,E1 4.1812,E2 246.1417} C_DIS
LIN {X -129.8659,Y -58.8351,Z 182,A -151.3055,B 4.3185,C 0.2893,E1 4.1834,E2 244.2051} C_DIS
LIN {X -127.9927,Y -62.8028,Z 182,A -149.5514,B 4.3182,C 0.2938,E1 4.1855,E2 242.453} C_DIS
LIN {X -126.2853,Y -66.1686,Z 182,A -148.0469,B 4.318,C 0.2977,E1 4.1874,E2 240.9508} C_DIS
LIN {X -124.3235,Y -69.7889,Z 182,A -146.2542,B 4.3178,C 0.3007,E1 4.1899,E2 239.1401} C_DIS
LIN {X -121.9878,Y -73.7956,Z 182,A -144.3298,B 4.3175,C 0.3047,E1 4.1926,E2 237.2082} C_DIS
LIN {X -119.514,Y -77.7383,Z 182,A -142.4562,B 4.3172,C 0.309,E1 4.1955,E2 235.3349} C_DIS
LIN {X -117.0656,Y -81.3785,Z 182,A -140.601,B 4.3169,C 0.3124,E1 4.1984,E2 233.4677} C_DIS
LIN {X -114.3346,Y -85.1729,Z 182,A -138.6701,B 4.3167,C 0.3161,E1 4.2016,E2 231.5304} C_DIS
LIN {X -111.4991,Y -88.8525,Z 182,A -136.7469,B 4.3164,C 0.3197,E1 4.2049,E2 229.6} C_DIS
LIN {X -108.47,Y -92.5264,Z 182,A -134.8515,B 4.3161,C 0.3239,E1 4.2083,E2 227.7077} C_DIS
LIN {X -105.6345,Y -95.7506,Z 182,A -133.0247,B 4.3159,C 0.3266,E1 4.2117,E2 225.8674} C_DIS
LIN {X -102.4448,Y -99.1558,Z 182,A -131.1062,B 4.3156,C 0.33,E1 4.2154,E2 223.9434} C_DIS
LIN {X -99.0933,Y -102.5054,Z 182,A -129.1707,B 4.3154,C 0.3334,E1 4.2193,E2 222.0039} C_DIS
LIN {X -95.7555,Y -105.6301,Z 182,A -127.2725,B 4.3151,C 0.3362,E1 4.2232,E2 220.0976} C_DIS
LIN {X -92.2317,Y -108.7205,Z 182,A -125.4052,B 4.3149,C 0.3397,E1 4.2272,E2 218.2328} C_DIS
LIN {X -89.0863,Y -111.3131,Z 182,A -123.7084,B 4.3147,C 0.342,E1 4.2309,E2 216.5281} C_DIS
LIN {X -85.6181,Y -114.0021,Z 182,A -121.9284,B 4.3145,C 0.3447,E1 4.2348,E2 214.746} C_DIS
LIN {X -82.0872,Y -116.5698,Z 182,A -120.0947,B 4.3143,C 0.3467,E1 4.239,E2 212.9015} C_DIS
LIN {X -78.2326,Y -119.1911,Z 182,A -118.2458,B 4.3141,C 0.3497,E1 4.2433,E2 211.056} C_DIS
LIN {X -74.7871,Y -121.3828,Z 182,A -116.5566,B 4.3139,C 0.3516,E1 4.2473,E2 209.3601} C_DIS
LIN {X -71.032,Y -123.6183,Z 182,A -114.7042,B 4.3139,C 0.353,E1 4.2518,E2 207.4945} C_DIS
LIN {X -67.1863,Y -125.7495,Z 182,A -112.9042,B 4.3136,C 0.3549,E1 4.2563,E2 205.6898} C_DIS
LIN {X -63.3113,Y -127.7419,Z 182,A -111.2055,B 4.3134,C 0.3574,E1 4.2605,E2 203.9981} C_DIS
LIN {X -60.1652,Y -129.2537,Z 182,A -109.8474,B 4.3133,C 0.3594,E1 4.2639,E2 202.6459} C_DIS
LIN {X -56.7118,Y -130.8054,Z 182,A -108.2088,B 4.3133,C 0.3598,E1 4.2681,E2 200.991} C_DIS
LIN {X -52.9339,Y -132.3798,Z 182,A -106.5573,B 4.3131,C 0.3613,E1 4.2724,E2 199.3383} C_DIS
LIN {X -49.0785,Y -133.8588,Z 182,A -104.9659,B 4.3129,C 0.3634,E1 4.2765,E2 197.7561} C_DIS
LIN {X -45.7907,Y -135.0189,Z 182,A -103.5513,B 4.3129,C 0.3644,E1 4.2803,E2 196.3393} C_DIS
LIN {X -41.947,Y -136.26,Z 182,A -101.8103,B 4.3129,C 0.3644,E1 4.285,E2 194.5816} C_DIS
LIN {X -37.4392,Y -137.5687,Z 182,A -100.0072,B 4.3127,C 0.3665,E1 4.2898,E2 192.7897} C_DIS
LIN {X -34.0551,Y -138.445,Z 182,A -98.5921,B 4.3127,C 0.3671,E1 4.2936,E2 191.3727} C_DIS
LIN {X -30.1058,Y -139.3555,Z 182,A -96.8835,B 4.3127,C 0.3671,E1 4.2983,E2 189.6526} C_DIS
LIN {X -25.5134,Y -140.2696,Z 182,A -95.2349,B 4.3124,C 0.3702,E1 4.3028,E2 188.0356} C_DIS
LIN {X -22.6382,Y -140.7641,Z 182,A -93.8801,B 4.3124,C 0.3688,E1 4.3066,E2 186.6553} C_DIS
LIN {X -18.5904,Y -141.3533,Z 182,A -92.3965,B 4.3124,C 0.3708,E1 4.3106,E2 185.1931} C_DIS
LIN {X -15.711,Y -141.703,Z 182,A -91.0657,B 4.3124,C 0.3694,E1 4.3144,E2 183.8391} C_DIS
LIN {X -11.6403,Y -142.0951,Z 182,A -89.4384,B 4.3124,C 0.3697,E1 4.3189,E2 182.2134} C_DIS
LIN {X -8.1401,Y -142.3395,Z 182,A -87.8956,B 4.3125,C 0.3684,E1 4.3232,E2 180.6516} C_DIS
LIN {X -4.647,Y -142.4966,Z 182,A -86.4785,B 4.3125,C 0.3682,E1 4.3272,E2 179.2323} C_DIS
LIN {X 0.0019,Y -142.5729,Z 182,A -84.5959,B 4.3125,C 0.3679,E1 4.3325,E2 177.3469} C_DIS
LIN {X 0.0019,Y -142.5729,Z 182,A -84.5959,B 4.3125,C 0.3679,E1 4.3325,E2 177.3469} C_DIS
Enddeposition()
LIN {X 0.9678,Y -133.6282,Z 183,A -84.9434,B 4.4528,C 0.3545,E1 4.471,E2 177.4358} C_DIS
Startdeposition()
$VEL.CP = VEL_PRINT
LIN {X -1.6605,Y -133.6245,Z 183,A -86.4727,B 4.4525,C 0.3586,E1 4.4666,E2 179.0168} C_DIS
LIN {X -4.9308,Y -133.5429,Z 183,A -87.7817,B 4.4525,C 0.3578,E1 4.463,E2 180.3146} C_DIS
LIN {X -7.8925,Y -133.4007,Z 183,A -89.0896,B 4.4525,C 0.3581,E1 4.4593,E2 181.6277} C_DIS
LIN {X -11.1563,Y -133.167,Z 183,A -90.5833,B 4.4525,C 0.3589,E1 4.4551,E2 183.1335} C_DIS
LIN {X -14.7244,Y -132.8205,Z 183,A -92.0642,B 4.4525,C 0.3581,E1 4.451,E2 184.6079} C_DIS
LIN {X -17.9938,Y -132.418,Z 183,A -93.4646,B 4.4525,C 0.3577,E1 4.4471,E2 186.0073} C_DIS
LIN {X -20.9274,Y -131.9855,Z 183,A -94.7567,B 4.4526,C 0.3575,E1 4.4436,E2 187.3025} C_DIS
Enddeposition()
END
